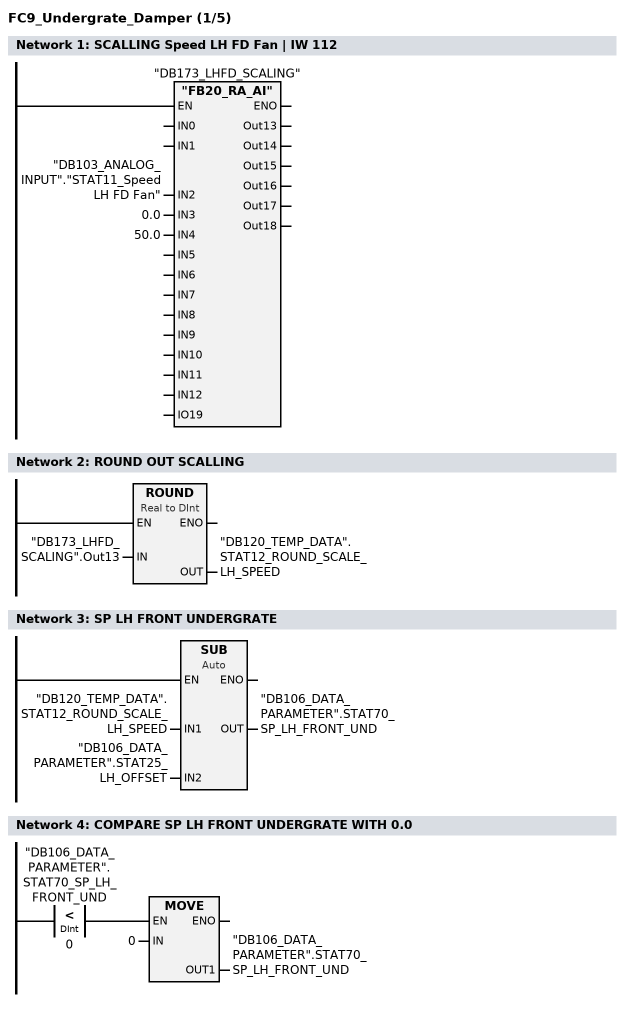
   RUNG wire#powerrail
      "DB173_LHFD_SCALING"(IN0 :=, IN1 :=, IN2 := "DB103_ANALOG_INPUT"."STAT11_Speed LH FD Fan", IN3 := 0.0, IN4 := 50.0, IN5 :=, IN6 :=, IN7 :=, IN8 :=, IN9 :=, IN10 :=, IN11 :=, IN12 :=, Out13 =>, IO19 :=, Out14 =>, Out15 =>, Out16 =>, Out17 =>, Out18 =>)
   END_RUNG
   // the same network as SCL:
   "DB173_LHFD_SCALING"(IN2 := "DB103_ANALOG_INPUT"."STAT11_Speed LH FD Fan", IN3 := 0.0, IN4 := 50.0);   // "FB20_RA_AI"
END_REGION

REGION Network 2: ROUND OUT SCALLING
   RUNG wire#powerrail
      { S7_Templates := "[SrcType := Real, DestType := DInt]" } Round(in := "DB173_LHFD_SCALING".Out13, out => "DB120_TEMP_DATA".STAT12_ROUND_SCALE_LH_SPEED)
   END_RUNG
   // the same network as SCL:
   "DB120_TEMP_DATA".STAT12_ROUND_SCALE_LH_SPEED := ROUND("DB173_LHFD_SCALING".Out13);
END_REGION

REGION Network 3: SP LH FRONT UNDERGRATE
   RUNG wire#powerrail
      Sub(in1 := "DB120_TEMP_DATA".STAT12_ROUND_SCALE_LH_SPEED, in2 := "DB106_DATA_PARAMETER".STAT25_LH_OFFSET, out => "DB106_DATA_PARAMETER".STAT70_SP_LH_FRONT_UND)
   END_RUNG
   // the same network as SCL:
   "DB106_DATA_PARAMETER".STAT70_SP_LH_FRONT_UND := "DB120_TEMP_DATA".STAT12_ROUND_SCALE_LH_SPEED - "DB106_DATA_PARAMETER".STAT25_LH_OFFSET;
END_REGION

REGION Network 4: COMPARE SP LH FRONT UNDERGRATE WITH 0.0
   RUNG wire#powerrail
      { S7_Templates := "SrcType := DInt" } LT_Contact(in1 := "DB106_DATA_PARAMETER".STAT70_SP_LH_FRONT_UND, in2 := 0)
      Move(in := 0, out1 => "DB106_DATA_PARAMETER".STAT70_SP_LH_FRONT_UND)
   END_RUNG
   // the same network as SCL:
   IF "DB106_DATA_PARAMETER".STAT70_SP_LH_FRONT_UND < 0 THEN
       "DB106_DATA_PARAMETER".STAT70_SP_LH_FRONT_UND := 0;
   END_IF;
END_REGION

REGION Network 5: LH FRONT UNDERGRATE POSITION | IW 208
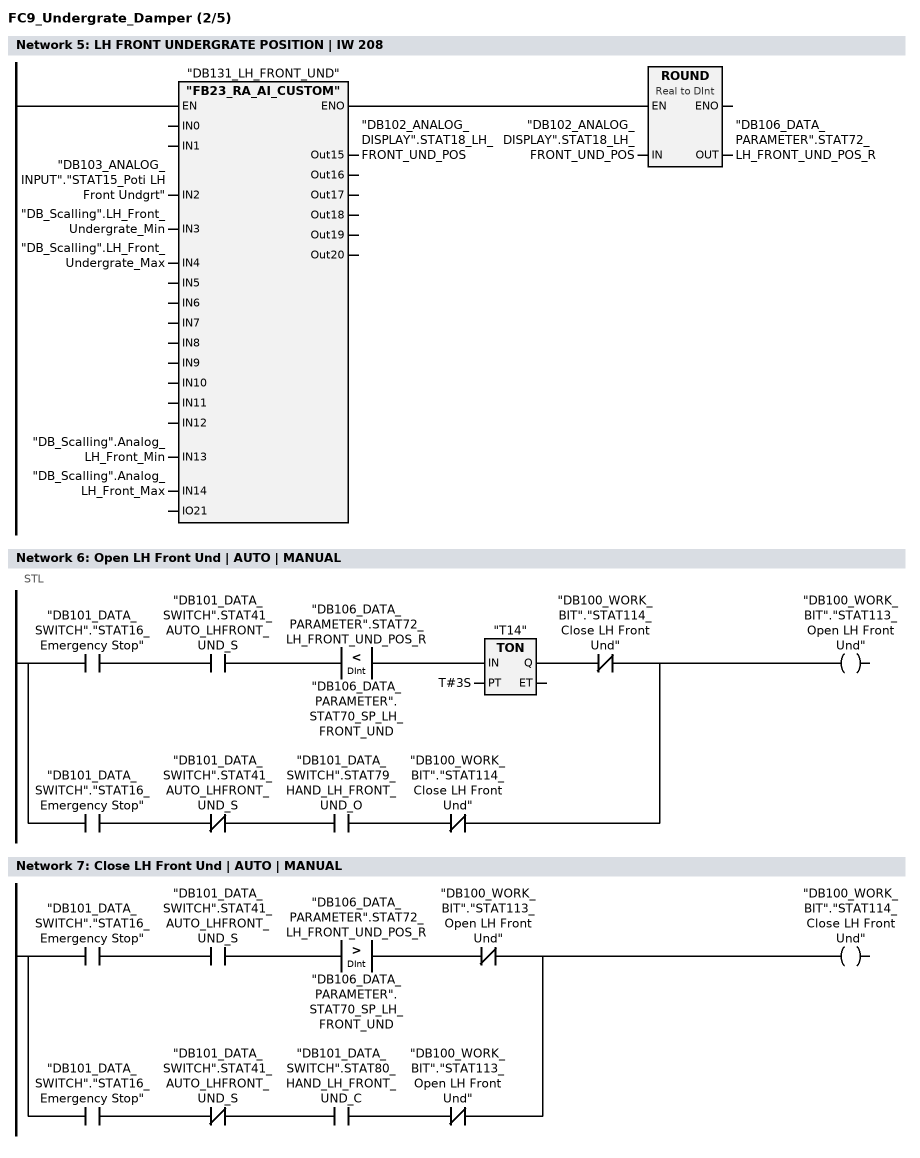
   RUNG wire#powerrail
      "DB131_LH_FRONT_UND"(IN0 :=, IN1 :=, IN2 := "DB103_ANALOG_INPUT"."STAT15_Poti LH Front Undgrt", IN3 := "DB_Scalling".LH_Front_Undergrate_Min, IN4 := "DB_Scalling".LH_Front_Undergrate_Max, IN5 :=, IN6 :=, IN7 :=, IN8 :=, IN9 :=, IN10 :=, IN11 :=, IN12 :=, IN13 := "DB_Scalling".Analog_LH_Front_Min, IN14 := "DB_Scalling".Analog_LH_Front_Max, IO21 :=, Out15 => "DB102_ANALOG_DISPLAY".STAT18_LH_FRONT_UND_POS, Out16 =>, Out17 =>, Out18 =>, Out19 =>, Out20 =>)
      { S7_Templates := "[SrcType := Real, DestType := DInt]" } Round(in := "DB102_ANALOG_DISPLAY".STAT18_LH_FRONT_UND_POS, out => "DB106_DATA_PARAMETER".STAT72_LH_FRONT_UND_POS_R)
   END_RUNG
   // the same network as SCL:
   "DB131_LH_FRONT_UND"(IN2 := "DB103_ANALOG_INPUT"."STAT15_Poti LH Front Undgrt",   // "FB23_RA_AI_CUSTOM"
                        IN3 := "DB_Scalling".LH_Front_Undergrate_Min,
                        IN4 := "DB_Scalling".LH_Front_Undergrate_Max,
                        IN13 := "DB_Scalling".Analog_LH_Front_Min,
                        IN14 := "DB_Scalling".Analog_LH_Front_Max,
                        Out15 => "DB102_ANALOG_DISPLAY".STAT18_LH_FRONT_UND_POS,
                        ENO => #_w1);
   IF #_w1 THEN
       "DB106_DATA_PARAMETER".STAT72_LH_FRONT_UND_POS_R := ROUND("DB102_ANALOG_DISPLAY".STAT18_LH_FRONT_UND_POS);
   END_IF;
END_REGION

REGION Network 6: Open LH Front Und | AUTO | MANUAL
   // STL
   "T14".TON(IN := "DB101_DATA_SWITCH"."STAT16_Emergency Stop" AND "DB101_DATA_SWITCH".STAT41_AUTO_LHFRONT_UND_S AND ("DB106_DATA_PARAMETER".STAT72_LH_FRONT_UND_POS_R < "DB106_DATA_PARAMETER".STAT70_SP_LH_FRONT_UND),
             PT := T#3S);
   "DB100_WORK_BIT"."STAT113_Open LH Front Und" := ("T14".Q AND NOT "DB100_WORK_BIT"."STAT114_Close LH Front Und") OR ("DB101_DATA_SWITCH"."STAT16_Emergency Stop" AND NOT "DB101_DATA_SWITCH".STAT41_AUTO_LHFRONT_UND_S AND "DB101_DATA_SWITCH".STAT79_HAND_LH_FRONT_UND_O AND NOT "DB100_WORK_BIT"."STAT114_Close LH Front Und");
END_REGION

REGION Network 7: Close LH Front Und | AUTO | MANUAL
   RUNG wire#powerrail
      Contact( "DB101_DATA_SWITCH"."STAT16_Emergency Stop" )
      Contact( "DB101_DATA_SWITCH".STAT41_AUTO_LHFRONT_UND_S )
      { S7_Templates := "SrcType := DInt" } GT_Contact(in1 := "DB106_DATA_PARAMETER".STAT72_LH_FRONT_UND_POS_R, in2 := "DB106_DATA_PARAMETER".STAT70_SP_LH_FRONT_UND)
      I_Contact( "DB100_WORK_BIT"."STAT113_Open LH Front Und" )
      wire#w1
      Coil( "DB100_WORK_BIT"."STAT114_Close LH Front Und" )
   END_RUNG
   RUNG wire#powerrail
      Contact( "DB101_DATA_SWITCH"."STAT16_Emergency Stop" )
      I_Contact( "DB101_DATA_SWITCH".STAT41_AUTO_LHFRONT_UND_S )
      Contact( "DB101_DATA_SWITCH".STAT80_HAND_LH_FRONT_UND_C )
      I_Contact( "DB100_WORK_BIT"."STAT113_Open LH Front Und" )
   END_RUNG wire#w1
   // the same network as SCL:
   "DB100_WORK_BIT"."STAT114_Close LH Front Und" := ("DB101_DATA_SWITCH"."STAT16_Emergency Stop" AND "DB101_DATA_SWITCH".STAT41_AUTO_LHFRONT_UND_S AND ("DB106_DATA_PARAMETER".STAT72_LH_FRONT_UND_POS_R > "DB106_DATA_PARAMETER".STAT70_SP_LH_FRONT_UND) AND NOT "DB100_WORK_BIT"."STAT113_Open LH Front Und") OR ("DB101_DATA_SWITCH"."STAT16_Emergency Stop" AND NOT "DB101_DATA_SWITCH".STAT41_AUTO_LHFRONT_UND_S AND "DB101_DATA_SWITCH".STAT80_HAND_LH_FRONT_UND_C AND NOT "DB100_WORK_BIT"."STAT113_Open LH Front Und");
END_REGION

REGION Network 8: SCALLING Speed RH FD Fan | IW 114
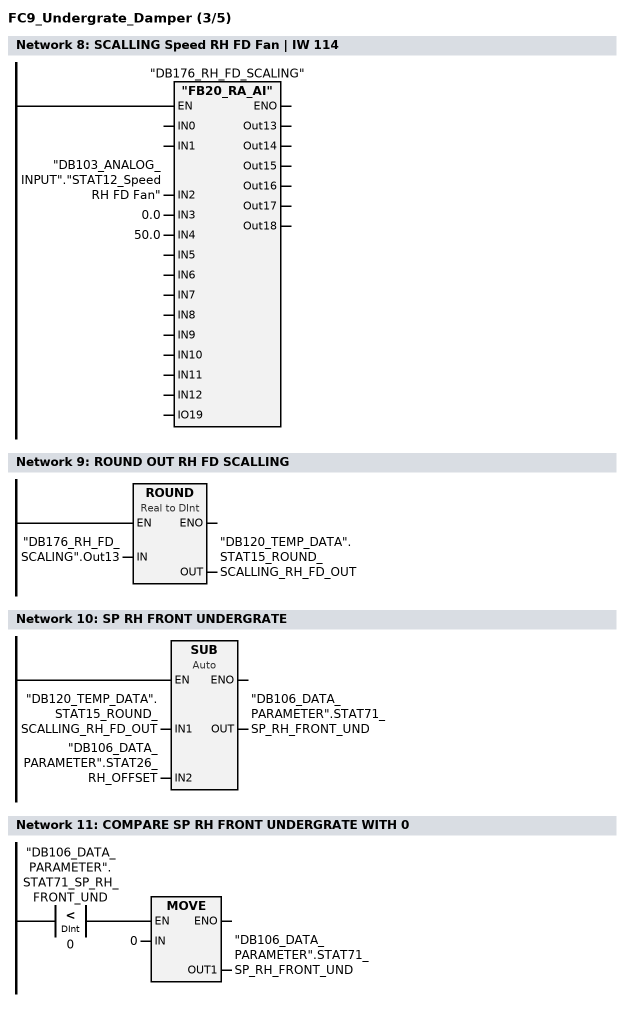
   RUNG wire#powerrail
      "DB176_RH_FD_SCALING"(IN0 :=, IN1 :=, IN2 := "DB103_ANALOG_INPUT"."STAT12_Speed RH FD Fan", IN3 := 0.0, IN4 := 50.0, IN5 :=, IN6 :=, IN7 :=, IN8 :=, IN9 :=, IN10 :=, IN11 :=, IN12 :=, Out13 =>, IO19 :=, Out14 =>, Out15 =>, Out16 =>, Out17 =>, Out18 =>)
   END_RUNG
   // the same network as SCL:
   "DB176_RH_FD_SCALING"(IN2 := "DB103_ANALOG_INPUT"."STAT12_Speed RH FD Fan", IN3 := 0.0, IN4 := 50.0);   // "FB20_RA_AI"
END_REGION

REGION Network 9: ROUND OUT RH FD SCALLING
   RUNG wire#powerrail
      { S7_Templates := "[SrcType := Real, DestType := DInt]" } Round(in := "DB176_RH_FD_SCALING".Out13, out => "DB120_TEMP_DATA".STAT15_ROUND_SCALLING_RH_FD_OUT)
   END_RUNG
   // the same network as SCL:
   "DB120_TEMP_DATA".STAT15_ROUND_SCALLING_RH_FD_OUT := ROUND("DB176_RH_FD_SCALING".Out13);
END_REGION

REGION Network 10: SP RH FRONT UNDERGRATE
   RUNG wire#powerrail
      Sub(in1 := "DB120_TEMP_DATA".STAT15_ROUND_SCALLING_RH_FD_OUT, in2 := "DB106_DATA_PARAMETER".STAT26_RH_OFFSET, out => "DB106_DATA_PARAMETER".STAT71_SP_RH_FRONT_UND)
   END_RUNG
   // the same network as SCL:
   "DB106_DATA_PARAMETER".STAT71_SP_RH_FRONT_UND := "DB120_TEMP_DATA".STAT15_ROUND_SCALLING_RH_FD_OUT - "DB106_DATA_PARAMETER".STAT26_RH_OFFSET;
END_REGION

REGION Network 11: COMPARE SP RH FRONT UNDERGRATE WITH 0
   RUNG wire#powerrail
      { S7_Templates := "SrcType := DInt" } LT_Contact(in1 := "DB106_DATA_PARAMETER".STAT71_SP_RH_FRONT_UND, in2 := 0)
      Move(in := 0, out1 => "DB106_DATA_PARAMETER".STAT71_SP_RH_FRONT_UND)
   END_RUNG
   // the same network as SCL:
   IF "DB106_DATA_PARAMETER".STAT71_SP_RH_FRONT_UND < 0 THEN
       "DB106_DATA_PARAMETER".STAT71_SP_RH_FRONT_UND := 0;
   END_IF;
END_REGION

REGION Network 12: Poti RH Front Undgrt(FEED BACK POSITION) RH FRONT UNDERGRATE
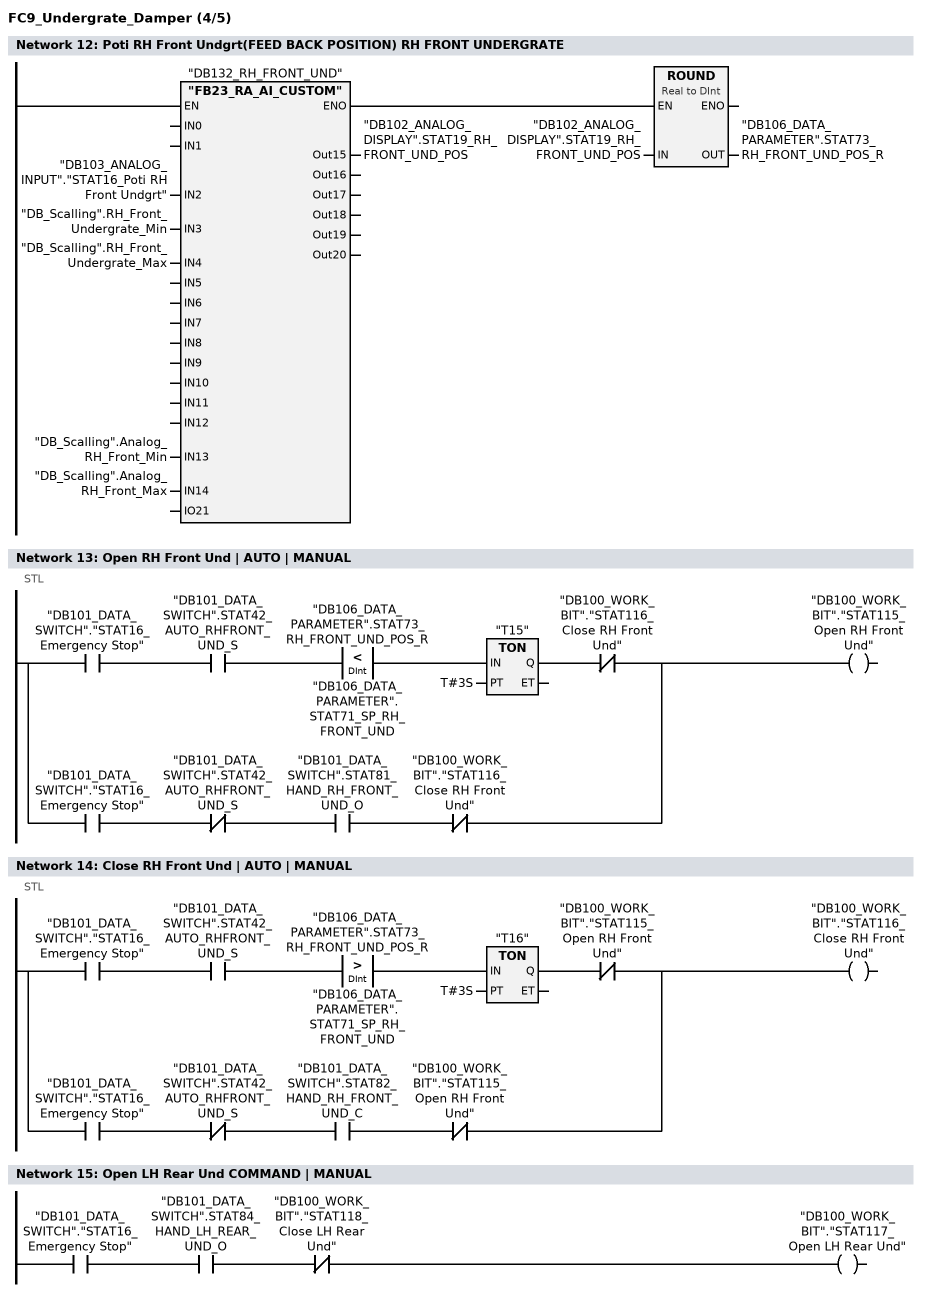
   RUNG wire#powerrail
      "DB132_RH_FRONT_UND"(IN0 :=, IN1 :=, IN2 := "DB103_ANALOG_INPUT"."STAT16_Poti RH Front Undgrt", IN3 := "DB_Scalling".RH_Front_Undergrate_Min, IN4 := "DB_Scalling".RH_Front_Undergrate_Max, IN5 :=, IN6 :=, IN7 :=, IN8 :=, IN9 :=, IN10 :=, IN11 :=, IN12 :=, IN13 := "DB_Scalling".Analog_RH_Front_Min, IN14 := "DB_Scalling".Analog_RH_Front_Max, IO21 :=, Out15 => "DB102_ANALOG_DISPLAY".STAT19_RH_FRONT_UND_POS, Out16 =>, Out17 =>, Out18 =>, Out19 =>, Out20 =>)
      { S7_Templates := "[SrcType := Real, DestType := DInt]" } Round(in := "DB102_ANALOG_DISPLAY".STAT19_RH_FRONT_UND_POS, out => "DB106_DATA_PARAMETER".STAT73_RH_FRONT_UND_POS_R)
   END_RUNG
   // the same network as SCL:
   "DB132_RH_FRONT_UND"(IN2 := "DB103_ANALOG_INPUT"."STAT16_Poti RH Front Undgrt",   // "FB23_RA_AI_CUSTOM"
                        IN3 := "DB_Scalling".RH_Front_Undergrate_Min,
                        IN4 := "DB_Scalling".RH_Front_Undergrate_Max,
                        IN13 := "DB_Scalling".Analog_RH_Front_Min,
                        IN14 := "DB_Scalling".Analog_RH_Front_Max,
                        Out15 => "DB102_ANALOG_DISPLAY".STAT19_RH_FRONT_UND_POS,
                        ENO => #_w1);
   IF #_w1 THEN
       "DB106_DATA_PARAMETER".STAT73_RH_FRONT_UND_POS_R := ROUND("DB102_ANALOG_DISPLAY".STAT19_RH_FRONT_UND_POS);
   END_IF;
END_REGION

REGION Network 13: Open RH Front Und | AUTO | MANUAL
   // STL
   "T15".TON(IN := "DB101_DATA_SWITCH"."STAT16_Emergency Stop" AND "DB101_DATA_SWITCH".STAT42_AUTO_RHFRONT_UND_S AND ("DB106_DATA_PARAMETER".STAT73_RH_FRONT_UND_POS_R < "DB106_DATA_PARAMETER".STAT71_SP_RH_FRONT_UND),
             PT := T#3S);
   "DB100_WORK_BIT"."STAT115_Open RH Front Und" := ("T15".Q AND NOT "DB100_WORK_BIT"."STAT116_Close RH Front Und") OR ("DB101_DATA_SWITCH"."STAT16_Emergency Stop" AND NOT "DB101_DATA_SWITCH".STAT42_AUTO_RHFRONT_UND_S AND "DB101_DATA_SWITCH".STAT81_HAND_RH_FRONT_UND_O AND NOT "DB100_WORK_BIT"."STAT116_Close RH Front Und");
END_REGION

REGION Network 14: Close RH Front Und | AUTO | MANUAL
   // STL
   "T16".TON(IN := "DB101_DATA_SWITCH"."STAT16_Emergency Stop" AND "DB101_DATA_SWITCH".STAT42_AUTO_RHFRONT_UND_S AND ("DB106_DATA_PARAMETER".STAT73_RH_FRONT_UND_POS_R > "DB106_DATA_PARAMETER".STAT71_SP_RH_FRONT_UND),
             PT := T#3S);
   "DB100_WORK_BIT"."STAT116_Close RH Front Und" := ("T16".Q AND NOT "DB100_WORK_BIT"."STAT115_Open RH Front Und") OR ("DB101_DATA_SWITCH"."STAT16_Emergency Stop" AND NOT "DB101_DATA_SWITCH".STAT42_AUTO_RHFRONT_UND_S AND "DB101_DATA_SWITCH".STAT82_HAND_RH_FRONT_UND_C AND NOT "DB100_WORK_BIT"."STAT115_Open RH Front Und");
END_REGION

REGION Network 15: Open LH Rear Und COMMAND | MANUAL
   RUNG wire#powerrail
      Contact( "DB101_DATA_SWITCH"."STAT16_Emergency Stop" )
      Contact( "DB101_DATA_SWITCH".STAT84_HAND_LH_REAR_UND_O )
      I_Contact( "DB100_WORK_BIT"."STAT118_Close LH Rear Und" )
      Coil( "DB100_WORK_BIT"."STAT117_Open LH Rear Und" )
   END_RUNG
   // the same network as SCL:
   "DB100_WORK_BIT"."STAT117_Open LH Rear Und" := "DB101_DATA_SWITCH"."STAT16_Emergency Stop" AND "DB101_DATA_SWITCH".STAT84_HAND_LH_REAR_UND_O AND NOT "DB100_WORK_BIT"."STAT118_Close LH Rear Und";
END_REGION

REGION Network 16: Close LH Rear Und COMMAND | MANUAL
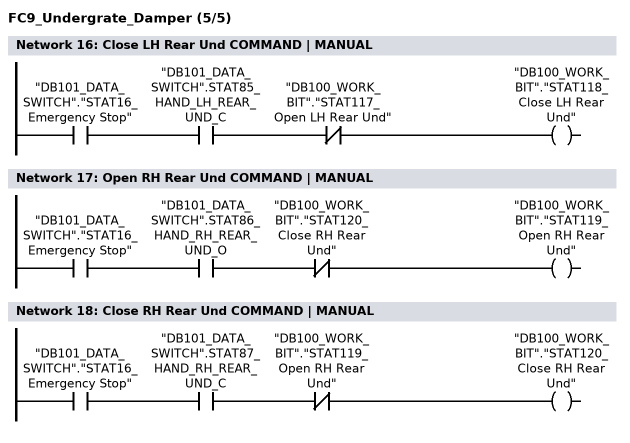
   RUNG wire#powerrail
      Contact( "DB101_DATA_SWITCH"."STAT16_Emergency Stop" )
      Contact( "DB101_DATA_SWITCH".STAT85_HAND_LH_REAR_UND_C )
      I_Contact( "DB100_WORK_BIT"."STAT117_Open LH Rear Und" )
      Coil( "DB100_WORK_BIT"."STAT118_Close LH Rear Und" )
   END_RUNG
   // the same network as SCL:
   "DB100_WORK_BIT"."STAT118_Close LH Rear Und" := "DB101_DATA_SWITCH"."STAT16_Emergency Stop" AND "DB101_DATA_SWITCH".STAT85_HAND_LH_REAR_UND_C AND NOT "DB100_WORK_BIT"."STAT117_Open LH Rear Und";
END_REGION

REGION Network 17: Open RH Rear Und COMMAND | MANUAL
   RUNG wire#powerrail
      Contact( "DB101_DATA_SWITCH"."STAT16_Emergency Stop" )
      Contact( "DB101_DATA_SWITCH".STAT86_HAND_RH_REAR_UND_O )
      I_Contact( "DB100_WORK_BIT"."STAT120_Close RH Rear Und" )
      Coil( "DB100_WORK_BIT"."STAT119_Open RH Rear Und" )
   END_RUNG
   // the same network as SCL:
   "DB100_WORK_BIT"."STAT119_Open RH Rear Und" := "DB101_DATA_SWITCH"."STAT16_Emergency Stop" AND "DB101_DATA_SWITCH".STAT86_HAND_RH_REAR_UND_O AND NOT "DB100_WORK_BIT"."STAT120_Close RH Rear Und";
END_REGION

REGION Network 18: Close RH Rear Und COMMAND | MANUAL
   RUNG wire#powerrail
      Contact( "DB101_DATA_SWITCH"."STAT16_Emergency Stop" )
      Contact( "DB101_DATA_SWITCH".STAT87_HAND_RH_REAR_UND_C )
      I_Contact( "DB100_WORK_BIT"."STAT119_Open RH Rear Und" )
      Coil( "DB100_WORK_BIT"."STAT120_Close RH Rear Und" )
   END_RUNG
   // the same network as SCL:
   "DB100_WORK_BIT"."STAT120_Close RH Rear Und" := "DB101_DATA_SWITCH"."STAT16_Emergency Stop" AND "DB101_DATA_SWITCH".STAT87_HAND_RH_REAR_UND_C AND NOT "DB100_WORK_BIT"."STAT119_Open RH Rear Und";
END_REGION
END_FUNCTION

FUNCTION "FC10_COAL_COUNTER" : Void   // FC10, LAD
TITLE = COAL COUNTER
{ S7_Optimized_Access := 'TRUE' }
VERSION : 0.1
BEGIN

REGION Network 1: LH TOTAL COAL
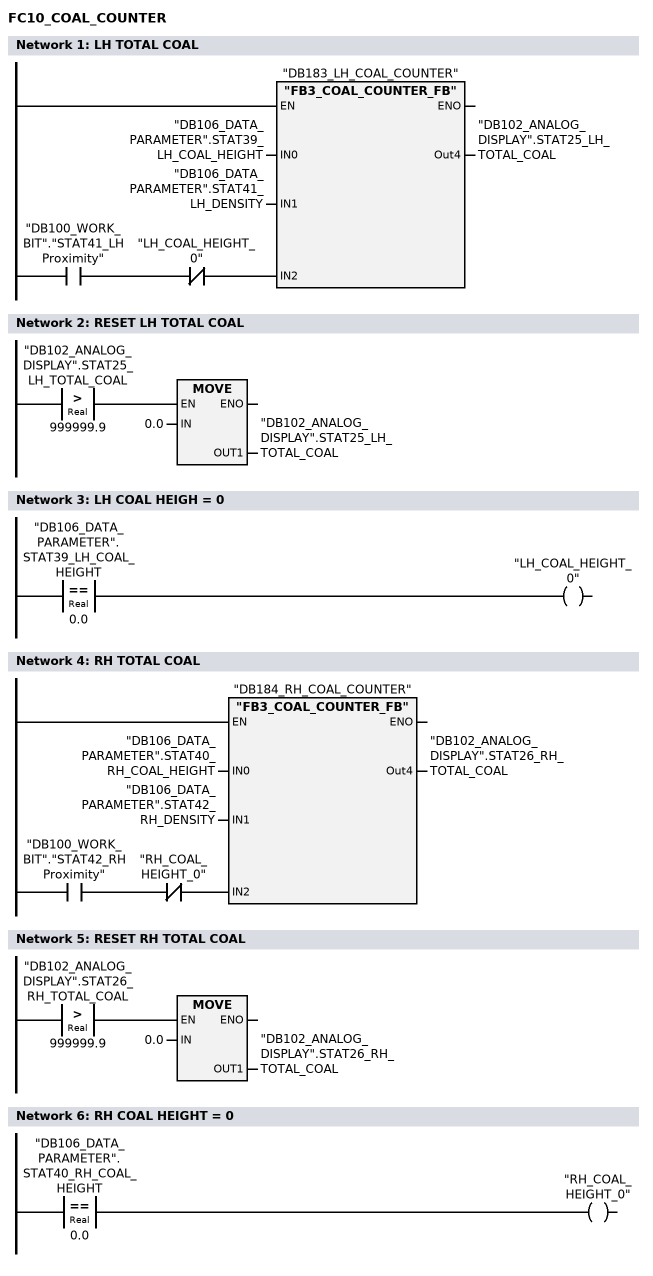
   RUNG wire#powerrail
      "DB183_LH_COAL_COUNTER"(IN2 := wire#w1, IN0 := "DB106_DATA_PARAMETER".STAT39_LH_COAL_HEIGHT, IN1 := "DB106_DATA_PARAMETER".STAT41_LH_DENSITY, Out4 => "DB102_ANALOG_DISPLAY".STAT25_LH_TOTAL_COAL)
   END_RUNG
   RUNG wire#powerrail
      Contact( "DB100_WORK_BIT"."STAT41_LH Proximity" )
      I_Contact( "LH_COAL_HEIGHT_0" )
   END_RUNG wire#w1
   // the same network as SCL:
   "DB183_LH_COAL_COUNTER"(IN0 := "DB106_DATA_PARAMETER".STAT39_LH_COAL_HEIGHT,   // "FB3_COAL_COUNTER_FB"
                           IN1 := "DB106_DATA_PARAMETER".STAT41_LH_DENSITY,
                           IN2 := "DB100_WORK_BIT"."STAT41_LH Proximity" AND NOT "LH_COAL_HEIGHT_0",
                           Out4 => "DB102_ANALOG_DISPLAY".STAT25_LH_TOTAL_COAL);
END_REGION

REGION Network 2: RESET LH TOTAL COAL
   RUNG wire#powerrail
      { S7_Templates := "SrcType := Real" } GT_Contact(in1 := "DB102_ANALOG_DISPLAY".STAT25_LH_TOTAL_COAL, in2 := 999999.9)
      Move(in := 0.0, out1 => "DB102_ANALOG_DISPLAY".STAT25_LH_TOTAL_COAL)
   END_RUNG
   // the same network as SCL:
   IF "DB102_ANALOG_DISPLAY".STAT25_LH_TOTAL_COAL > 999999.9 THEN
       "DB102_ANALOG_DISPLAY".STAT25_LH_TOTAL_COAL := 0.0;
   END_IF;
END_REGION

REGION Network 3: LH COAL HEIGH = 0
   RUNG wire#powerrail
      { S7_Templates := "SrcType := Real" } EQ_Contact(in1 := "DB106_DATA_PARAMETER".STAT39_LH_COAL_HEIGHT, in2 := 0.0)
      Coil( "LH_COAL_HEIGHT_0" )
   END_RUNG
   // the same network as SCL:
   "LH_COAL_HEIGHT_0" := "DB106_DATA_PARAMETER".STAT39_LH_COAL_HEIGHT = 0.0;
END_REGION

REGION Network 4: RH TOTAL COAL
   RUNG wire#powerrail
      "DB184_RH_COAL_COUNTER"(IN2 := wire#w1, IN0 := "DB106_DATA_PARAMETER".STAT40_RH_COAL_HEIGHT, IN1 := "DB106_DATA_PARAMETER".STAT42_RH_DENSITY, Out4 => "DB102_ANALOG_DISPLAY".STAT26_RH_TOTAL_COAL)
   END_RUNG
   RUNG wire#powerrail
      Contact( "DB100_WORK_BIT"."STAT42_RH Proximity" )
      I_Contact( "RH_COAL_HEIGHT_0" )
   END_RUNG wire#w1
   // the same network as SCL:
   "DB184_RH_COAL_COUNTER"(IN0 := "DB106_DATA_PARAMETER".STAT40_RH_COAL_HEIGHT,   // "FB3_COAL_COUNTER_FB"
                           IN1 := "DB106_DATA_PARAMETER".STAT42_RH_DENSITY,
                           IN2 := "DB100_WORK_BIT"."STAT42_RH Proximity" AND NOT "RH_COAL_HEIGHT_0",
                           Out4 => "DB102_ANALOG_DISPLAY".STAT26_RH_TOTAL_COAL);
END_REGION

REGION Network 5: RESET RH TOTAL COAL
   RUNG wire#powerrail
      { S7_Templates := "SrcType := Real" } GT_Contact(in1 := "DB102_ANALOG_DISPLAY".STAT26_RH_TOTAL_COAL, in2 := 999999.9)
      Move(in := 0.0, out1 => "DB102_ANALOG_DISPLAY".STAT26_RH_TOTAL_COAL)
   END_RUNG
   // the same network as SCL:
   IF "DB102_ANALOG_DISPLAY".STAT26_RH_TOTAL_COAL > 999999.9 THEN
       "DB102_ANALOG_DISPLAY".STAT26_RH_TOTAL_COAL := 0.0;
   END_IF;
END_REGION

REGION Network 6: RH COAL HEIGHT = 0
   RUNG wire#powerrail
      { S7_Templates := "SrcType := Real" } EQ_Contact(in1 := "DB106_DATA_PARAMETER".STAT40_RH_COAL_HEIGHT, in2 := 0.0)
      Coil( "RH_COAL_HEIGHT_0" )
   END_RUNG
   // the same network as SCL:
   "RH_COAL_HEIGHT_0" := "DB106_DATA_PARAMETER".STAT40_RH_COAL_HEIGHT = 0.0;
END_REGION
END_FUNCTION

FUNCTION "FC11_Alarm" : Void   // FC11, LAD
TITLE = ALARM
{ S7_Optimized_Access := 'TRUE' }
VERSION : 0.1
BEGIN

REGION Network 1: Alarm Low Water PreWarning
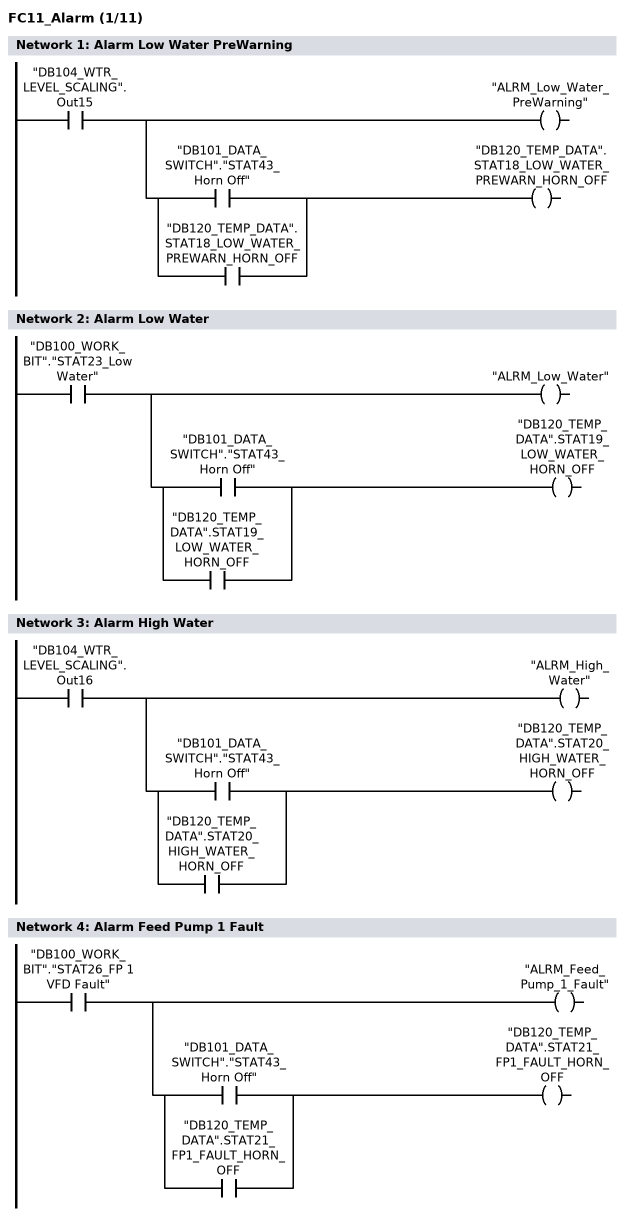
   RUNG wire#powerrail
      Contact( "DB104_WTR_LEVEL_SCALING".Out15 )
      wire#w1
      Coil( "ALRM_Low_Water_PreWarning" )
   END_RUNG
   RUNG wire#w1
      Contact( "DB101_DATA_SWITCH"."STAT43_Horn Off" )
      wire#w2
      Coil( "DB120_TEMP_DATA".STAT18_LOW_WATER_PREWARN_HORN_OFF )
   END_RUNG
   RUNG wire#w1
      Contact( "DB120_TEMP_DATA".STAT18_LOW_WATER_PREWARN_HORN_OFF )
   END_RUNG wire#w2
   // the same network as SCL:
   "ALRM_Low_Water_PreWarning" := "DB104_WTR_LEVEL_SCALING".Out15;
   "DB120_TEMP_DATA".STAT18_LOW_WATER_PREWARN_HORN_OFF := "DB104_WTR_LEVEL_SCALING".Out15 AND ("DB101_DATA_SWITCH"."STAT43_Horn Off" OR "DB120_TEMP_DATA".STAT18_LOW_WATER_PREWARN_HORN_OFF);
END_REGION

REGION Network 2: Alarm Low Water
   RUNG wire#powerrail
      Contact( "DB100_WORK_BIT"."STAT23_Low Water" )
      wire#w1
      Coil( "ALRM_Low_Water" )
   END_RUNG
   RUNG wire#w1
      Contact( "DB101_DATA_SWITCH"."STAT43_Horn Off" )
      wire#w2
      Coil( "DB120_TEMP_DATA".STAT19_LOW_WATER_HORN_OFF )
   END_RUNG
   RUNG wire#w1
      Contact( "DB120_TEMP_DATA".STAT19_LOW_WATER_HORN_OFF )
   END_RUNG wire#w2
   // the same network as SCL:
   "ALRM_Low_Water" := "DB100_WORK_BIT"."STAT23_Low Water";
   "DB120_TEMP_DATA".STAT19_LOW_WATER_HORN_OFF := "DB100_WORK_BIT"."STAT23_Low Water" AND ("DB101_DATA_SWITCH"."STAT43_Horn Off" OR "DB120_TEMP_DATA".STAT19_LOW_WATER_HORN_OFF);
END_REGION

REGION Network 3: Alarm High Water
   RUNG wire#powerrail
      Contact( "DB104_WTR_LEVEL_SCALING".Out16 )
      wire#w1
      Coil( "ALRM_High_Water" )
   END_RUNG
   RUNG wire#w1
      Contact( "DB101_DATA_SWITCH"."STAT43_Horn Off" )
      wire#w2
      Coil( "DB120_TEMP_DATA".STAT20_HIGH_WATER_HORN_OFF )
   END_RUNG
   RUNG wire#w1
      Contact( "DB120_TEMP_DATA".STAT20_HIGH_WATER_HORN_OFF )
   END_RUNG wire#w2
   // the same network as SCL:
   "ALRM_High_Water" := "DB104_WTR_LEVEL_SCALING".Out16;
   "DB120_TEMP_DATA".STAT20_HIGH_WATER_HORN_OFF := "DB104_WTR_LEVEL_SCALING".Out16 AND ("DB101_DATA_SWITCH"."STAT43_Horn Off" OR "DB120_TEMP_DATA".STAT20_HIGH_WATER_HORN_OFF);
END_REGION

REGION Network 4: Alarm Feed Pump 1 Fault
   RUNG wire#powerrail
      Contact( "DB100_WORK_BIT"."STAT26_FP 1 VFD Fault" )
      wire#w1
      Coil( "ALRM_Feed_Pump_1_Fault" )
   END_RUNG
   RUNG wire#w1
      Contact( "DB101_DATA_SWITCH"."STAT43_Horn Off" )
      wire#w2
      Coil( "DB120_TEMP_DATA".STAT21_FP1_FAULT_HORN_OFF )
   END_RUNG
   RUNG wire#w1
      Contact( "DB120_TEMP_DATA".STAT21_FP1_FAULT_HORN_OFF )
   END_RUNG wire#w2
   // the same network as SCL:
   "ALRM_Feed_Pump_1_Fault" := "DB100_WORK_BIT"."STAT26_FP 1 VFD Fault";
   "DB120_TEMP_DATA".STAT21_FP1_FAULT_HORN_OFF := "DB100_WORK_BIT"."STAT26_FP 1 VFD Fault" AND ("DB101_DATA_SWITCH"."STAT43_Horn Off" OR "DB120_TEMP_DATA".STAT21_FP1_FAULT_HORN_OFF);
END_REGION

REGION Network 5: Alarm Feed Pump 2 Fault
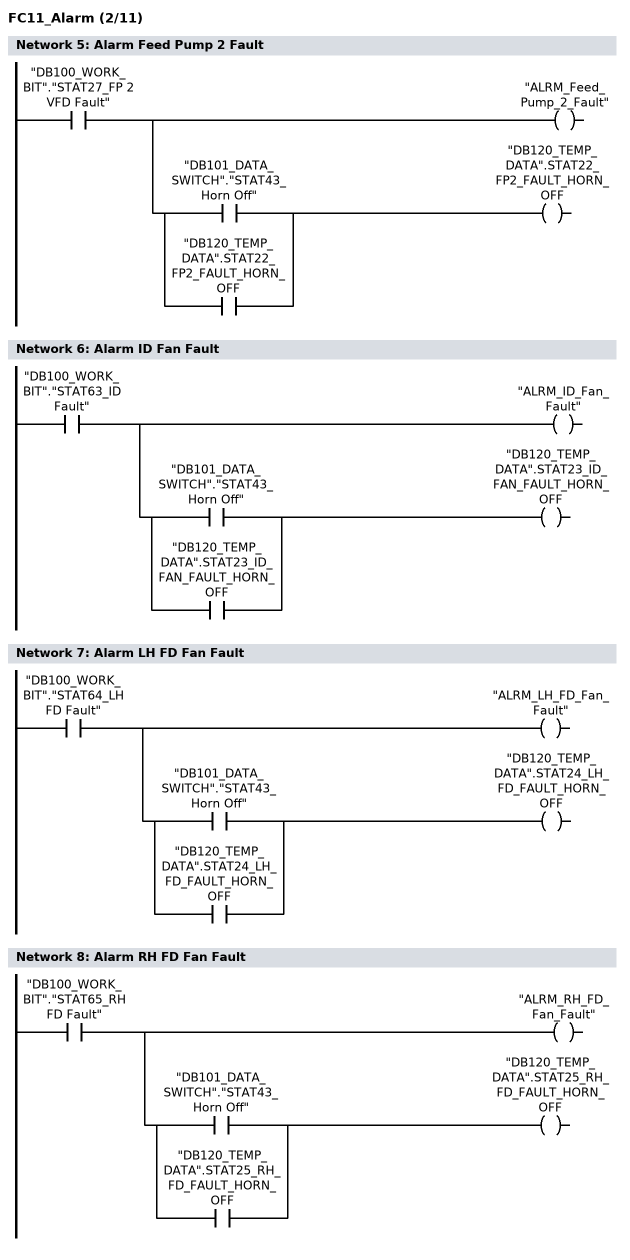
   RUNG wire#powerrail
      Contact( "DB100_WORK_BIT"."STAT27_FP 2 VFD Fault" )
      wire#w1
      Coil( "ALRM_Feed_Pump_2_Fault" )
   END_RUNG
   RUNG wire#w1
      Contact( "DB101_DATA_SWITCH"."STAT43_Horn Off" )
      wire#w2
      Coil( "DB120_TEMP_DATA".STAT22_FP2_FAULT_HORN_OFF )
   END_RUNG
   RUNG wire#w1
      Contact( "DB120_TEMP_DATA".STAT22_FP2_FAULT_HORN_OFF )
   END_RUNG wire#w2
   // the same network as SCL:
   "ALRM_Feed_Pump_2_Fault" := "DB100_WORK_BIT"."STAT27_FP 2 VFD Fault";
   "DB120_TEMP_DATA".STAT22_FP2_FAULT_HORN_OFF := "DB100_WORK_BIT"."STAT27_FP 2 VFD Fault" AND ("DB101_DATA_SWITCH"."STAT43_Horn Off" OR "DB120_TEMP_DATA".STAT22_FP2_FAULT_HORN_OFF);
END_REGION

REGION Network 6: Alarm ID Fan Fault
   RUNG wire#powerrail
      Contact( "DB100_WORK_BIT"."STAT63_ID Fault" )
      wire#w1
      Coil( "ALRM_ID_Fan_Fault" )
   END_RUNG
   RUNG wire#w1
      Contact( "DB101_DATA_SWITCH"."STAT43_Horn Off" )
      wire#w2
      Coil( "DB120_TEMP_DATA".STAT23_ID_FAN_FAULT_HORN_OFF )
   END_RUNG
   RUNG wire#w1
      Contact( "DB120_TEMP_DATA".STAT23_ID_FAN_FAULT_HORN_OFF )
   END_RUNG wire#w2
   // the same network as SCL:
   "ALRM_ID_Fan_Fault" := "DB100_WORK_BIT"."STAT63_ID Fault";
   "DB120_TEMP_DATA".STAT23_ID_FAN_FAULT_HORN_OFF := "DB100_WORK_BIT"."STAT63_ID Fault" AND ("DB101_DATA_SWITCH"."STAT43_Horn Off" OR "DB120_TEMP_DATA".STAT23_ID_FAN_FAULT_HORN_OFF);
END_REGION

REGION Network 7: Alarm LH FD Fan Fault
   RUNG wire#powerrail
      Contact( "DB100_WORK_BIT"."STAT64_LH FD Fault" )
      wire#w1
      Coil( "ALRM_LH_FD_Fan_Fault" )
   END_RUNG
   RUNG wire#w1
      Contact( "DB101_DATA_SWITCH"."STAT43_Horn Off" )
      wire#w2
      Coil( "DB120_TEMP_DATA".STAT24_LH_FD_FAULT_HORN_OFF )
   END_RUNG
   RUNG wire#w1
      Contact( "DB120_TEMP_DATA".STAT24_LH_FD_FAULT_HORN_OFF )
   END_RUNG wire#w2
   // the same network as SCL:
   "ALRM_LH_FD_Fan_Fault" := "DB100_WORK_BIT"."STAT64_LH FD Fault";
   "DB120_TEMP_DATA".STAT24_LH_FD_FAULT_HORN_OFF := "DB100_WORK_BIT"."STAT64_LH FD Fault" AND ("DB101_DATA_SWITCH"."STAT43_Horn Off" OR "DB120_TEMP_DATA".STAT24_LH_FD_FAULT_HORN_OFF);
END_REGION

REGION Network 8: Alarm RH FD Fan Fault
   RUNG wire#powerrail
      Contact( "DB100_WORK_BIT"."STAT65_RH FD Fault" )
      wire#w1
      Coil( "ALRM_RH_FD_Fan_Fault" )
   END_RUNG
   RUNG wire#w1
      Contact( "DB101_DATA_SWITCH"."STAT43_Horn Off" )
      wire#w2
      Coil( "DB120_TEMP_DATA".STAT25_RH_FD_FAULT_HORN_OFF )
   END_RUNG
   RUNG wire#w1
      Contact( "DB120_TEMP_DATA".STAT25_RH_FD_FAULT_HORN_OFF )
   END_RUNG wire#w2
   // the same network as SCL:
   "ALRM_RH_FD_Fan_Fault" := "DB100_WORK_BIT"."STAT65_RH FD Fault";
   "DB120_TEMP_DATA".STAT25_RH_FD_FAULT_HORN_OFF := "DB100_WORK_BIT"."STAT65_RH FD Fault" AND ("DB101_DATA_SWITCH"."STAT43_Horn Off" OR "DB120_TEMP_DATA".STAT25_RH_FD_FAULT_HORN_OFF);
END_REGION

REGION Network 9: Alarm LH Stoker Fault
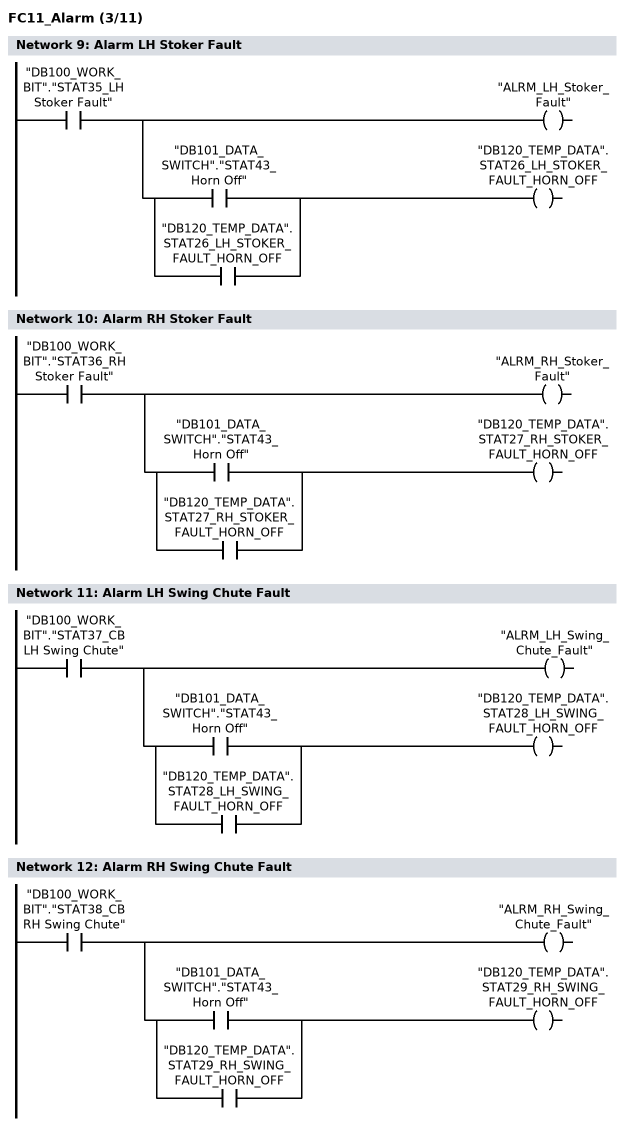
   RUNG wire#powerrail
      Contact( "DB100_WORK_BIT"."STAT35_LH Stoker Fault" )
      wire#w1
      Coil( "ALRM_LH_Stoker_Fault" )
   END_RUNG
   RUNG wire#w1
      Contact( "DB101_DATA_SWITCH"."STAT43_Horn Off" )
      wire#w2
      Coil( "DB120_TEMP_DATA".STAT26_LH_STOKER_FAULT_HORN_OFF )
   END_RUNG
   RUNG wire#w1
      Contact( "DB120_TEMP_DATA".STAT26_LH_STOKER_FAULT_HORN_OFF )
   END_RUNG wire#w2
   // the same network as SCL:
   "ALRM_LH_Stoker_Fault" := "DB100_WORK_BIT"."STAT35_LH Stoker Fault";
   "DB120_TEMP_DATA".STAT26_LH_STOKER_FAULT_HORN_OFF := "DB100_WORK_BIT"."STAT35_LH Stoker Fault" AND ("DB101_DATA_SWITCH"."STAT43_Horn Off" OR "DB120_TEMP_DATA".STAT26_LH_STOKER_FAULT_HORN_OFF);
END_REGION

REGION Network 10: Alarm RH Stoker Fault
   RUNG wire#powerrail
      Contact( "DB100_WORK_BIT"."STAT36_RH Stoker Fault" )
      wire#w1
      Coil( "ALRM_RH_Stoker_Fault" )
   END_RUNG
   RUNG wire#w1
      Contact( "DB101_DATA_SWITCH"."STAT43_Horn Off" )
      wire#w2
      Coil( "DB120_TEMP_DATA".STAT27_RH_STOKER_FAULT_HORN_OFF )
   END_RUNG
   RUNG wire#w1
      Contact( "DB120_TEMP_DATA".STAT27_RH_STOKER_FAULT_HORN_OFF )
   END_RUNG wire#w2
   // the same network as SCL:
   "ALRM_RH_Stoker_Fault" := "DB100_WORK_BIT"."STAT36_RH Stoker Fault";
   "DB120_TEMP_DATA".STAT27_RH_STOKER_FAULT_HORN_OFF := "DB100_WORK_BIT"."STAT36_RH Stoker Fault" AND ("DB101_DATA_SWITCH"."STAT43_Horn Off" OR "DB120_TEMP_DATA".STAT27_RH_STOKER_FAULT_HORN_OFF);
END_REGION

REGION Network 11: Alarm LH Swing Chute Fault
   RUNG wire#powerrail
      Contact( "DB100_WORK_BIT"."STAT37_CB LH Swing Chute" )
      wire#w1
      Coil( "ALRM_LH_Swing_Chute_Fault" )
   END_RUNG
   RUNG wire#w1
      Contact( "DB101_DATA_SWITCH"."STAT43_Horn Off" )
      wire#w2
      Coil( "DB120_TEMP_DATA".STAT28_LH_SWING_FAULT_HORN_OFF )
   END_RUNG
   RUNG wire#w1
      Contact( "DB120_TEMP_DATA".STAT28_LH_SWING_FAULT_HORN_OFF )
   END_RUNG wire#w2
   // the same network as SCL:
   "ALRM_LH_Swing_Chute_Fault" := "DB100_WORK_BIT"."STAT37_CB LH Swing Chute";
   "DB120_TEMP_DATA".STAT28_LH_SWING_FAULT_HORN_OFF := "DB100_WORK_BIT"."STAT37_CB LH Swing Chute" AND ("DB101_DATA_SWITCH"."STAT43_Horn Off" OR "DB120_TEMP_DATA".STAT28_LH_SWING_FAULT_HORN_OFF);
END_REGION

REGION Network 12: Alarm RH Swing Chute Fault
   RUNG wire#powerrail
      Contact( "DB100_WORK_BIT"."STAT38_CB RH Swing Chute" )
      wire#w1
      Coil( "ALRM_RH_Swing_Chute_Fault" )
   END_RUNG
   RUNG wire#w1
      Contact( "DB101_DATA_SWITCH"."STAT43_Horn Off" )
      wire#w2
      Coil( "DB120_TEMP_DATA".STAT29_RH_SWING_FAULT_HORN_OFF )
   END_RUNG
   RUNG wire#w1
      Contact( "DB120_TEMP_DATA".STAT29_RH_SWING_FAULT_HORN_OFF )
   END_RUNG wire#w2
   // the same network as SCL:
   "ALRM_RH_Swing_Chute_Fault" := "DB100_WORK_BIT"."STAT38_CB RH Swing Chute";
   "DB120_TEMP_DATA".STAT29_RH_SWING_FAULT_HORN_OFF := "DB100_WORK_BIT"."STAT38_CB RH Swing Chute" AND ("DB101_DATA_SWITCH"."STAT43_Horn Off" OR "DB120_TEMP_DATA".STAT29_RH_SWING_FAULT_HORN_OFF);
END_REGION

REGION Network 13: Alarm RAV1 Fault ASH VALVE 1
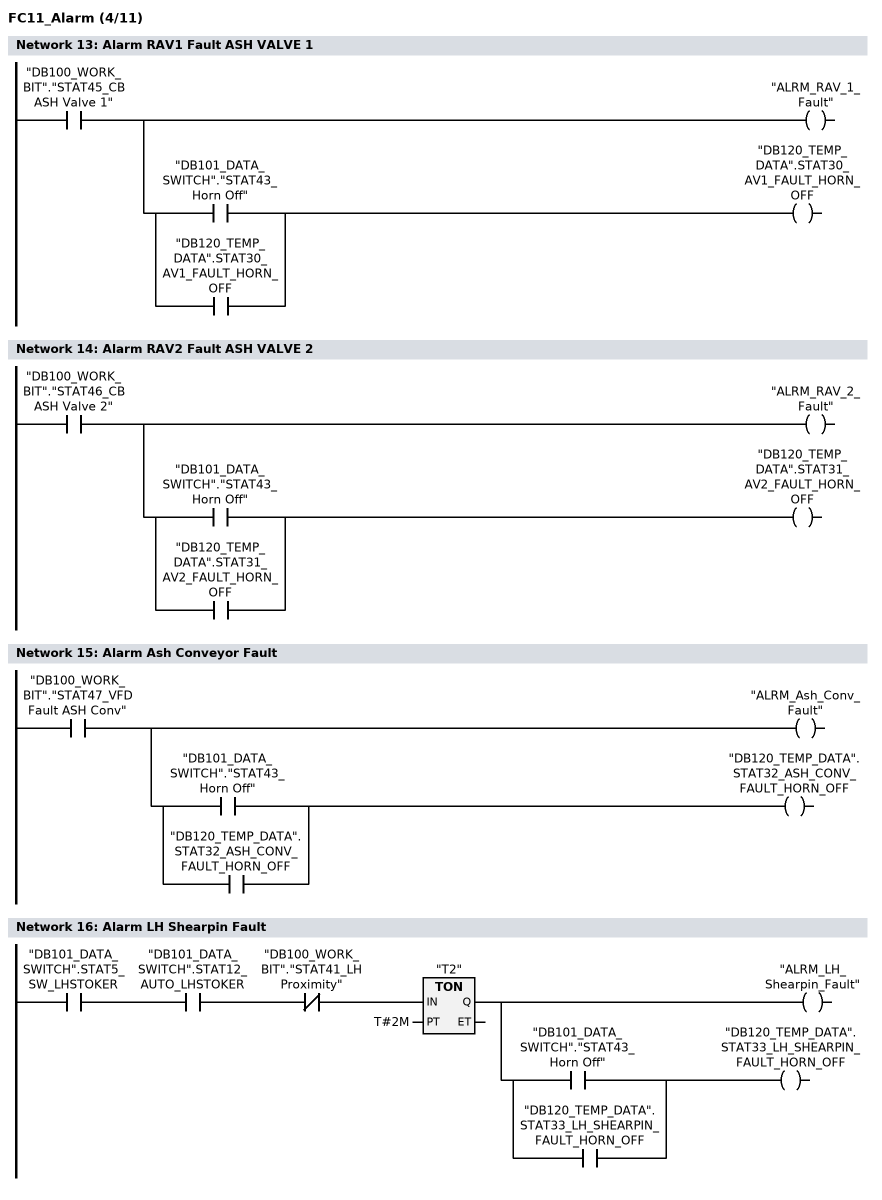
   RUNG wire#powerrail
      Contact( "DB100_WORK_BIT"."STAT45_CB ASH Valve 1" )
      wire#w1
      Coil( "ALRM_RAV_1_Fault" )
   END_RUNG
   RUNG wire#w1
      Contact( "DB101_DATA_SWITCH"."STAT43_Horn Off" )
      wire#w2
      Coil( "DB120_TEMP_DATA".STAT30_AV1_FAULT_HORN_OFF )
   END_RUNG
   RUNG wire#w1
      Contact( "DB120_TEMP_DATA".STAT30_AV1_FAULT_HORN_OFF )
   END_RUNG wire#w2
   // the same network as SCL:
   "ALRM_RAV_1_Fault" := "DB100_WORK_BIT"."STAT45_CB ASH Valve 1";
   "DB120_TEMP_DATA".STAT30_AV1_FAULT_HORN_OFF := "DB100_WORK_BIT"."STAT45_CB ASH Valve 1" AND ("DB101_DATA_SWITCH"."STAT43_Horn Off" OR "DB120_TEMP_DATA".STAT30_AV1_FAULT_HORN_OFF);
END_REGION

REGION Network 14: Alarm RAV2 Fault ASH VALVE 2
   RUNG wire#powerrail
      Contact( "DB100_WORK_BIT"."STAT46_CB ASH Valve 2" )
      wire#w1
      Coil( "ALRM_RAV_2_Fault" )
   END_RUNG
   RUNG wire#w1
      Contact( "DB101_DATA_SWITCH"."STAT43_Horn Off" )
      wire#w2
      Coil( "DB120_TEMP_DATA".STAT31_AV2_FAULT_HORN_OFF )
   END_RUNG
   RUNG wire#w1
      Contact( "DB120_TEMP_DATA".STAT31_AV2_FAULT_HORN_OFF )
   END_RUNG wire#w2
   // the same network as SCL:
   "ALRM_RAV_2_Fault" := "DB100_WORK_BIT"."STAT46_CB ASH Valve 2";
   "DB120_TEMP_DATA".STAT31_AV2_FAULT_HORN_OFF := "DB100_WORK_BIT"."STAT46_CB ASH Valve 2" AND ("DB101_DATA_SWITCH"."STAT43_Horn Off" OR "DB120_TEMP_DATA".STAT31_AV2_FAULT_HORN_OFF);
END_REGION

REGION Network 15: Alarm Ash Conveyor Fault
   RUNG wire#powerrail
      Contact( "DB100_WORK_BIT"."STAT47_VFD Fault ASH Conv" )
      wire#w1
      Coil( "ALRM_Ash_Conv_Fault" )
   END_RUNG
   RUNG wire#w1
      Contact( "DB101_DATA_SWITCH"."STAT43_Horn Off" )
      wire#w2
      Coil( "DB120_TEMP_DATA".STAT32_ASH_CONV_FAULT_HORN_OFF )
   END_RUNG
   RUNG wire#w1
      Contact( "DB120_TEMP_DATA".STAT32_ASH_CONV_FAULT_HORN_OFF )
   END_RUNG wire#w2
   // the same network as SCL:
   "ALRM_Ash_Conv_Fault" := "DB100_WORK_BIT"."STAT47_VFD Fault ASH Conv";
   "DB120_TEMP_DATA".STAT32_ASH_CONV_FAULT_HORN_OFF := "DB100_WORK_BIT"."STAT47_VFD Fault ASH Conv" AND ("DB101_DATA_SWITCH"."STAT43_Horn Off" OR "DB120_TEMP_DATA".STAT32_ASH_CONV_FAULT_HORN_OFF);
END_REGION

REGION Network 16: Alarm LH Shearpin Fault
   "T2".TON(IN := "DB101_DATA_SWITCH".STAT5_SW_LHSTOKER AND "DB101_DATA_SWITCH".STAT12_AUTO_LHSTOKER AND NOT "DB100_WORK_BIT"."STAT41_LH Proximity",
            PT := T#2M);
   "ALRM_LH_Shearpin_Fault" := "T2".Q;
   "DB120_TEMP_DATA".STAT33_LH_SHEARPIN_FAULT_HORN_OFF := "T2".Q AND ("DB101_DATA_SWITCH"."STAT43_Horn Off" OR "DB120_TEMP_DATA".STAT33_LH_SHEARPIN_FAULT_HORN_OFF);
END_REGION

REGION Network 17: Alarm RH Shearpin Fault
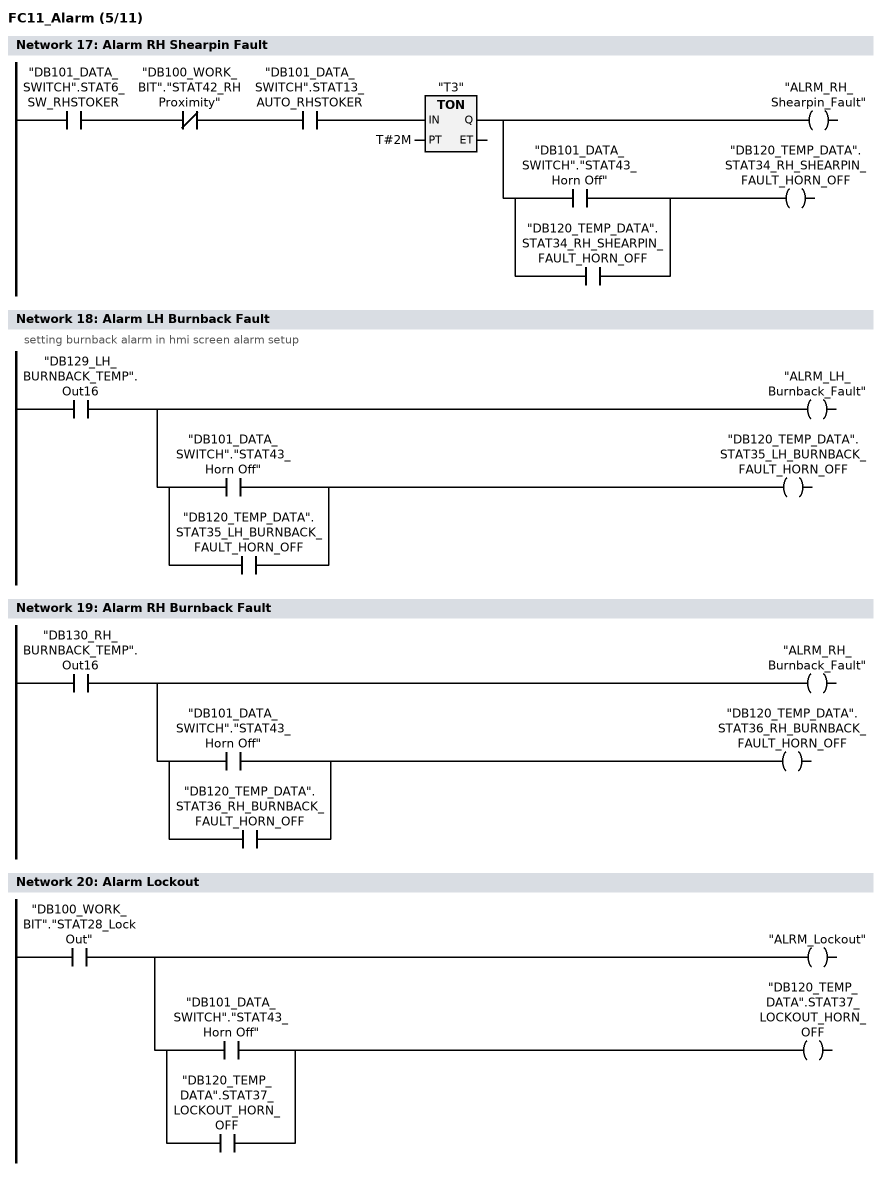
   "T3".TON(IN := "DB101_DATA_SWITCH".STAT6_SW_RHSTOKER AND NOT "DB100_WORK_BIT"."STAT42_RH Proximity" AND "DB101_DATA_SWITCH".STAT13_AUTO_RHSTOKER,
            PT := T#2M);
   "ALRM_RH_Shearpin_Fault" := "T3".Q;
   "DB120_TEMP_DATA".STAT34_RH_SHEARPIN_FAULT_HORN_OFF := "T3".Q AND ("DB101_DATA_SWITCH"."STAT43_Horn Off" OR "DB120_TEMP_DATA".STAT34_RH_SHEARPIN_FAULT_HORN_OFF);
END_REGION

REGION Network 18: Alarm LH Burnback Fault
   // setting burnback alarm in hmi screen alarm setup
   RUNG wire#powerrail
      Contact( "DB129_LH_BURNBACK_TEMP".Out16 )
      wire#w1
      Coil( "ALRM_LH_Burnback_Fault" )
   END_RUNG
   RUNG wire#w1
      Contact( "DB101_DATA_SWITCH"."STAT43_Horn Off" )
      wire#w2
      Coil( "DB120_TEMP_DATA".STAT35_LH_BURNBACK_FAULT_HORN_OFF )
   END_RUNG
   RUNG wire#w1
      Contact( "DB120_TEMP_DATA".STAT35_LH_BURNBACK_FAULT_HORN_OFF )
   END_RUNG wire#w2
   // the same network as SCL:
   "ALRM_LH_Burnback_Fault" := "DB129_LH_BURNBACK_TEMP".Out16;
   "DB120_TEMP_DATA".STAT35_LH_BURNBACK_FAULT_HORN_OFF := "DB129_LH_BURNBACK_TEMP".Out16 AND ("DB101_DATA_SWITCH"."STAT43_Horn Off" OR "DB120_TEMP_DATA".STAT35_LH_BURNBACK_FAULT_HORN_OFF);
END_REGION

REGION Network 19: Alarm RH Burnback Fault
   RUNG wire#powerrail
      Contact( "DB130_RH_BURNBACK_TEMP".Out16 )
      wire#w1
      Coil( "ALRM_RH_Burnback_Fault" )
   END_RUNG
   RUNG wire#w1
      Contact( "DB101_DATA_SWITCH"."STAT43_Horn Off" )
      wire#w2
      Coil( "DB120_TEMP_DATA".STAT36_RH_BURNBACK_FAULT_HORN_OFF )
   END_RUNG
   RUNG wire#w1
      Contact( "DB120_TEMP_DATA".STAT36_RH_BURNBACK_FAULT_HORN_OFF )
   END_RUNG wire#w2
   // the same network as SCL:
   "ALRM_RH_Burnback_Fault" := "DB130_RH_BURNBACK_TEMP".Out16;
   "DB120_TEMP_DATA".STAT36_RH_BURNBACK_FAULT_HORN_OFF := "DB130_RH_BURNBACK_TEMP".Out16 AND ("DB101_DATA_SWITCH"."STAT43_Horn Off" OR "DB120_TEMP_DATA".STAT36_RH_BURNBACK_FAULT_HORN_OFF);
END_REGION

REGION Network 20: Alarm Lockout
   RUNG wire#powerrail
      Contact( "DB100_WORK_BIT"."STAT28_Lock Out" )
      wire#w1
      Coil( "ALRM_Lockout" )
   END_RUNG
   RUNG wire#w1
      Contact( "DB101_DATA_SWITCH"."STAT43_Horn Off" )
      wire#w2
      Coil( "DB120_TEMP_DATA".STAT37_LOCKOUT_HORN_OFF )
   END_RUNG
   RUNG wire#w1
      Contact( "DB120_TEMP_DATA".STAT37_LOCKOUT_HORN_OFF )
   END_RUNG wire#w2
   // the same network as SCL:
   "ALRM_Lockout" := "DB100_WORK_BIT"."STAT28_Lock Out";
   "DB120_TEMP_DATA".STAT37_LOCKOUT_HORN_OFF := "DB100_WORK_BIT"."STAT28_Lock Out" AND ("DB101_DATA_SWITCH"."STAT43_Horn Off" OR "DB120_TEMP_DATA".STAT37_LOCKOUT_HORN_OFF);
END_REGION

REGION Network 21: Alarm Coal Hopper Low Level
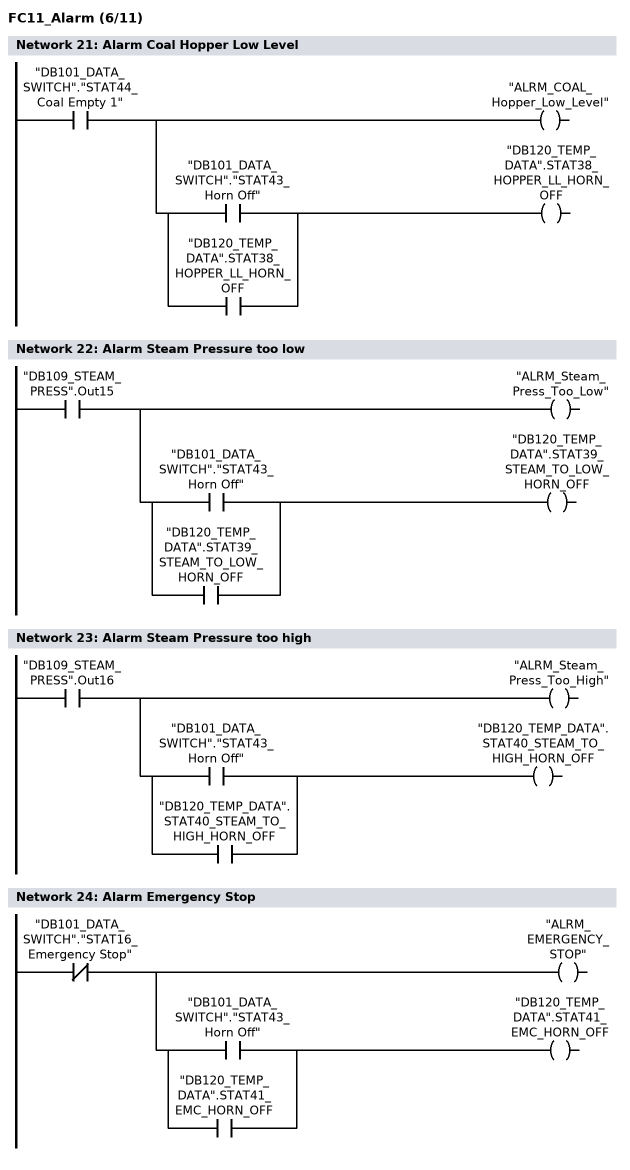
   RUNG wire#powerrail
      Contact( "DB101_DATA_SWITCH"."STAT44_Coal Empty 1" )
      wire#w1
      Coil( "ALRM_COAL_Hopper_Low_Level" )
   END_RUNG
   RUNG wire#w1
      Contact( "DB101_DATA_SWITCH"."STAT43_Horn Off" )
      wire#w2
      Coil( "DB120_TEMP_DATA".STAT38_HOPPER_LL_HORN_OFF )
   END_RUNG
   RUNG wire#w1
      Contact( "DB120_TEMP_DATA".STAT38_HOPPER_LL_HORN_OFF )
   END_RUNG wire#w2
   // the same network as SCL:
   "ALRM_COAL_Hopper_Low_Level" := "DB101_DATA_SWITCH"."STAT44_Coal Empty 1";
   "DB120_TEMP_DATA".STAT38_HOPPER_LL_HORN_OFF := "DB101_DATA_SWITCH"."STAT44_Coal Empty 1" AND ("DB101_DATA_SWITCH"."STAT43_Horn Off" OR "DB120_TEMP_DATA".STAT38_HOPPER_LL_HORN_OFF);
END_REGION

REGION Network 22: Alarm Steam Pressure too low
   RUNG wire#powerrail
      Contact( "DB109_STEAM_PRESS".Out15 )
      wire#w1
      Coil( "ALRM_Steam_Press_Too_Low" )
   END_RUNG
   RUNG wire#w1
      Contact( "DB101_DATA_SWITCH"."STAT43_Horn Off" )
      wire#w2
      Coil( "DB120_TEMP_DATA".STAT39_STEAM_TO_LOW_HORN_OFF )
   END_RUNG
   RUNG wire#w1
      Contact( "DB120_TEMP_DATA".STAT39_STEAM_TO_LOW_HORN_OFF )
   END_RUNG wire#w2
   // the same network as SCL:
   "ALRM_Steam_Press_Too_Low" := "DB109_STEAM_PRESS".Out15;
   "DB120_TEMP_DATA".STAT39_STEAM_TO_LOW_HORN_OFF := "DB109_STEAM_PRESS".Out15 AND ("DB101_DATA_SWITCH"."STAT43_Horn Off" OR "DB120_TEMP_DATA".STAT39_STEAM_TO_LOW_HORN_OFF);
END_REGION

REGION Network 23: Alarm Steam Pressure too high
   RUNG wire#powerrail
      Contact( "DB109_STEAM_PRESS".Out16 )
      wire#w1
      Coil( "ALRM_Steam_Press_Too_High" )
   END_RUNG
   RUNG wire#w1
      Contact( "DB101_DATA_SWITCH"."STAT43_Horn Off" )
      wire#w2
      Coil( "DB120_TEMP_DATA".STAT40_STEAM_TO_HIGH_HORN_OFF )
   END_RUNG
   RUNG wire#w1
      Contact( "DB120_TEMP_DATA".STAT40_STEAM_TO_HIGH_HORN_OFF )
   END_RUNG wire#w2
   // the same network as SCL:
   "ALRM_Steam_Press_Too_High" := "DB109_STEAM_PRESS".Out16;
   "DB120_TEMP_DATA".STAT40_STEAM_TO_HIGH_HORN_OFF := "DB109_STEAM_PRESS".Out16 AND ("DB101_DATA_SWITCH"."STAT43_Horn Off" OR "DB120_TEMP_DATA".STAT40_STEAM_TO_HIGH_HORN_OFF);
END_REGION

REGION Network 24: Alarm Emergency Stop
   RUNG wire#powerrail
      I_Contact( "DB101_DATA_SWITCH"."STAT16_Emergency Stop" )
      wire#w1
      Coil( "ALRM_EMERGENCY_STOP" )
   END_RUNG
   RUNG wire#w1
      Contact( "DB101_DATA_SWITCH"."STAT43_Horn Off" )
      wire#w2
      Coil( "DB120_TEMP_DATA".STAT41_EMC_HORN_OFF )
   END_RUNG
   RUNG wire#w1
      Contact( "DB120_TEMP_DATA".STAT41_EMC_HORN_OFF )
   END_RUNG wire#w2
   // the same network as SCL:
   "ALRM_EMERGENCY_STOP" := NOT "DB101_DATA_SWITCH"."STAT16_Emergency Stop";
   "DB120_TEMP_DATA".STAT41_EMC_HORN_OFF := NOT "DB101_DATA_SWITCH"."STAT16_Emergency Stop" AND ("DB101_DATA_SWITCH"."STAT43_Horn Off" OR "DB120_TEMP_DATA".STAT41_EMC_HORN_OFF);
END_REGION

REGION Network 25: Alarm Pump Pressure Low
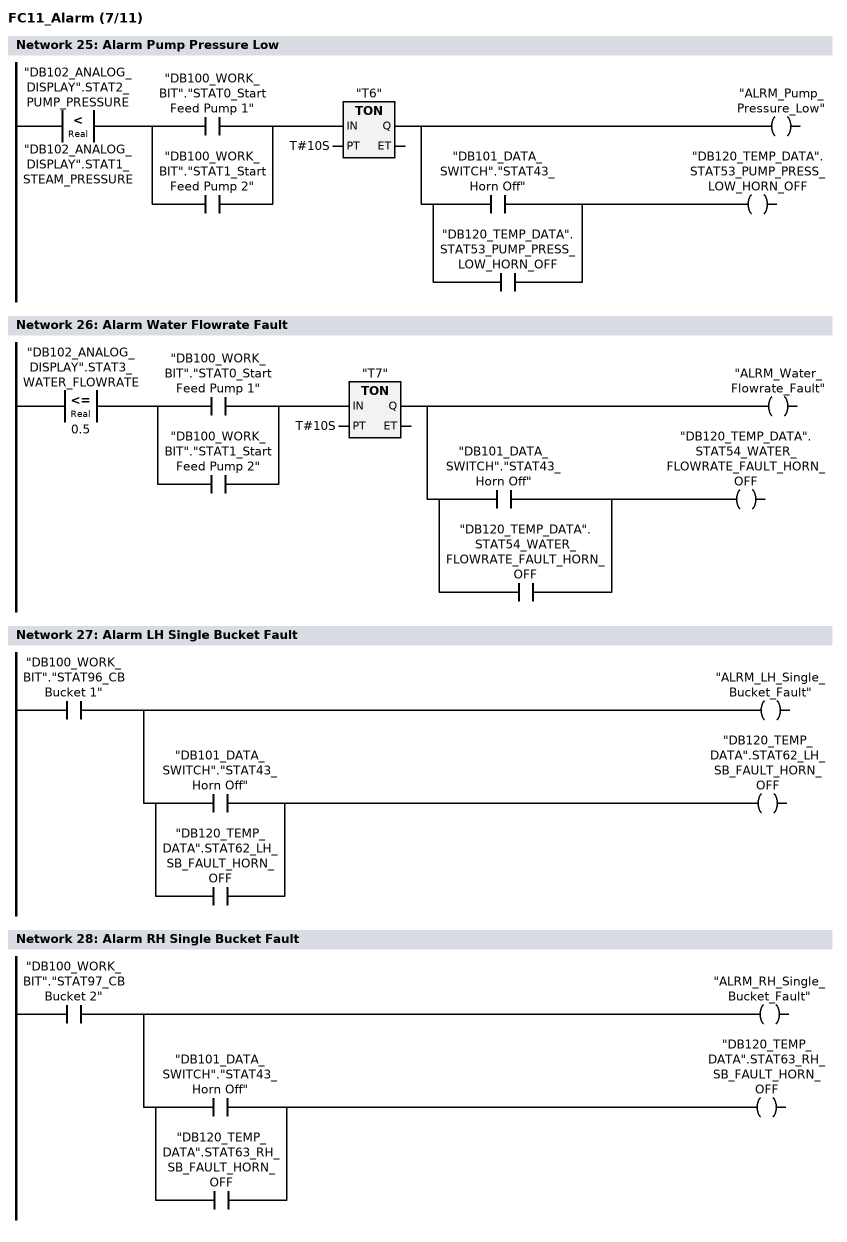
   "T6".TON(IN := ("DB102_ANALOG_DISPLAY".STAT2_PUMP_PRESSURE < "DB102_ANALOG_DISPLAY".STAT1_STEAM_PRESSURE) AND ("DB100_WORK_BIT"."STAT0_Start Feed Pump 1" OR "DB100_WORK_BIT"."STAT1_Start Feed Pump 2"),
            PT := T#10S);
   "ALRM_Pump_Pressure_Low" := "T6".Q;
   "DB120_TEMP_DATA".STAT53_PUMP_PRESS_LOW_HORN_OFF := "T6".Q AND ("DB101_DATA_SWITCH"."STAT43_Horn Off" OR "DB120_TEMP_DATA".STAT53_PUMP_PRESS_LOW_HORN_OFF);
END_REGION

REGION Network 26: Alarm Water Flowrate Fault
   "T7".TON(IN := ("DB102_ANALOG_DISPLAY".STAT3_WATER_FLOWRATE <= 0.5) AND ("DB100_WORK_BIT"."STAT0_Start Feed Pump 1" OR "DB100_WORK_BIT"."STAT1_Start Feed Pump 2"),
            PT := T#10S);
   "ALRM_Water_Flowrate_Fault" := "T7".Q;
   "DB120_TEMP_DATA".STAT54_WATER_FLOWRATE_FAULT_HORN_OFF := "T7".Q AND ("DB101_DATA_SWITCH"."STAT43_Horn Off" OR "DB120_TEMP_DATA".STAT54_WATER_FLOWRATE_FAULT_HORN_OFF);
END_REGION

REGION Network 27: Alarm LH Single Bucket Fault
   RUNG wire#powerrail
      Contact( "DB100_WORK_BIT"."STAT96_CB Bucket 1" )
      wire#w1
      Coil( "ALRM_LH_Single_Bucket_Fault" )
   END_RUNG
   RUNG wire#w1
      Contact( "DB101_DATA_SWITCH"."STAT43_Horn Off" )
      wire#w2
      Coil( "DB120_TEMP_DATA".STAT62_LH_SB_FAULT_HORN_OFF )
   END_RUNG
   RUNG wire#w1
      Contact( "DB120_TEMP_DATA".STAT62_LH_SB_FAULT_HORN_OFF )
   END_RUNG wire#w2
   // the same network as SCL:
   "ALRM_LH_Single_Bucket_Fault" := "DB100_WORK_BIT"."STAT96_CB Bucket 1";
   "DB120_TEMP_DATA".STAT62_LH_SB_FAULT_HORN_OFF := "DB100_WORK_BIT"."STAT96_CB Bucket 1" AND ("DB101_DATA_SWITCH"."STAT43_Horn Off" OR "DB120_TEMP_DATA".STAT62_LH_SB_FAULT_HORN_OFF);
END_REGION

REGION Network 28: Alarm RH Single Bucket Fault
   RUNG wire#powerrail
      Contact( "DB100_WORK_BIT"."STAT97_CB Bucket 2" )
      wire#w1
      Coil( "ALRM_RH_Single_Bucket_Fault" )
   END_RUNG
   RUNG wire#w1
      Contact( "DB101_DATA_SWITCH"."STAT43_Horn Off" )
      wire#w2
      Coil( "DB120_TEMP_DATA".STAT63_RH_SB_FAULT_HORN_OFF )
   END_RUNG
   RUNG wire#w1
      Contact( "DB120_TEMP_DATA".STAT63_RH_SB_FAULT_HORN_OFF )
   END_RUNG wire#w2
   // the same network as SCL:
   "ALRM_RH_Single_Bucket_Fault" := "DB100_WORK_BIT"."STAT97_CB Bucket 2";
   "DB120_TEMP_DATA".STAT63_RH_SB_FAULT_HORN_OFF := "DB100_WORK_BIT"."STAT97_CB Bucket 2" AND ("DB101_DATA_SWITCH"."STAT43_Horn Off" OR "DB120_TEMP_DATA".STAT63_RH_SB_FAULT_HORN_OFF);
END_REGION

REGION Network 29: Alarm FP Dry Run Protection
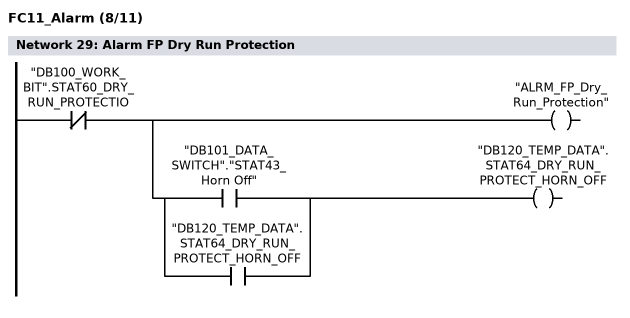
   RUNG wire#powerrail
      I_Contact( "DB100_WORK_BIT".STAT60_DRY_RUN_PROTECTIO )
      wire#w1
      Coil( "ALRM_FP_Dry_Run_Protection" )
   END_RUNG
   RUNG wire#w1
      Contact( "DB101_DATA_SWITCH"."STAT43_Horn Off" )
      wire#w2
      Coil( "DB120_TEMP_DATA".STAT64_DRY_RUN_PROTECT_HORN_OFF )
   END_RUNG
   RUNG wire#w1
      Contact( "DB120_TEMP_DATA".STAT64_DRY_RUN_PROTECT_HORN_OFF )
   END_RUNG wire#w2
   // the same network as SCL:
   "ALRM_FP_Dry_Run_Protection" := NOT "DB100_WORK_BIT".STAT60_DRY_RUN_PROTECTIO;
   "DB120_TEMP_DATA".STAT64_DRY_RUN_PROTECT_HORN_OFF := NOT "DB100_WORK_BIT".STAT60_DRY_RUN_PROTECTIO AND ("DB101_DATA_SWITCH"."STAT43_Horn Off" OR "DB120_TEMP_DATA".STAT64_DRY_RUN_PROTECT_HORN_OFF);
END_REGION

REGION Network 30: Alarm Horn
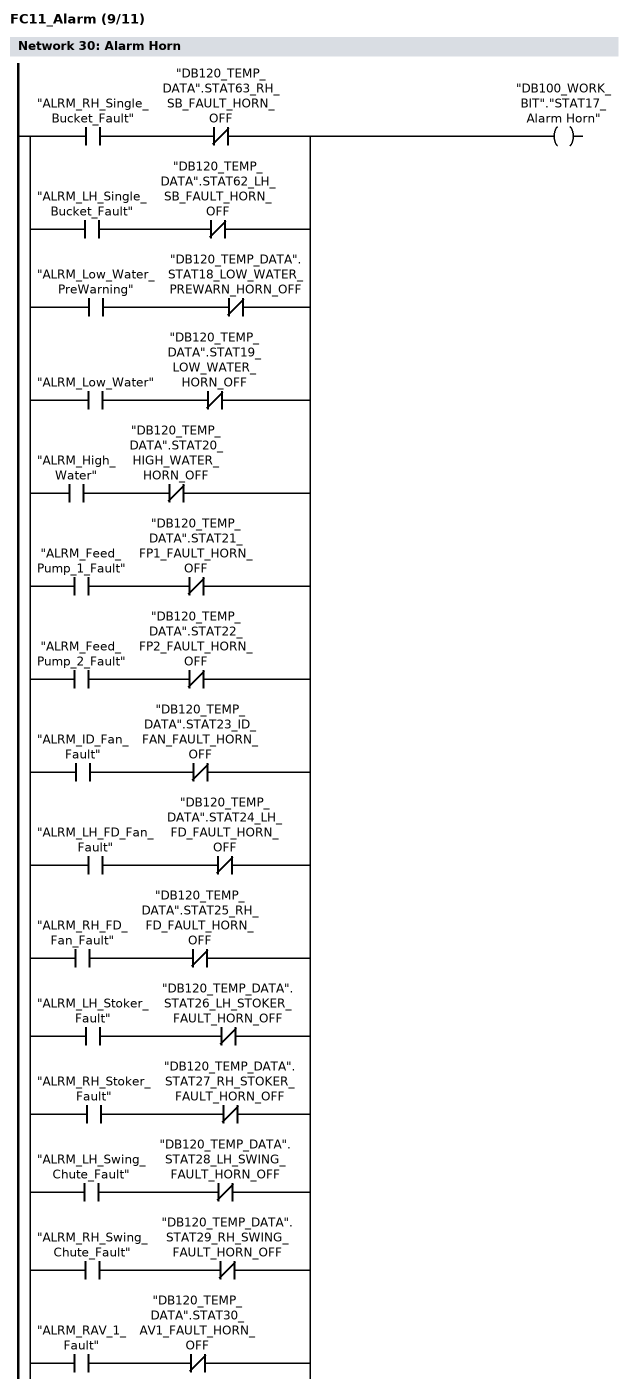
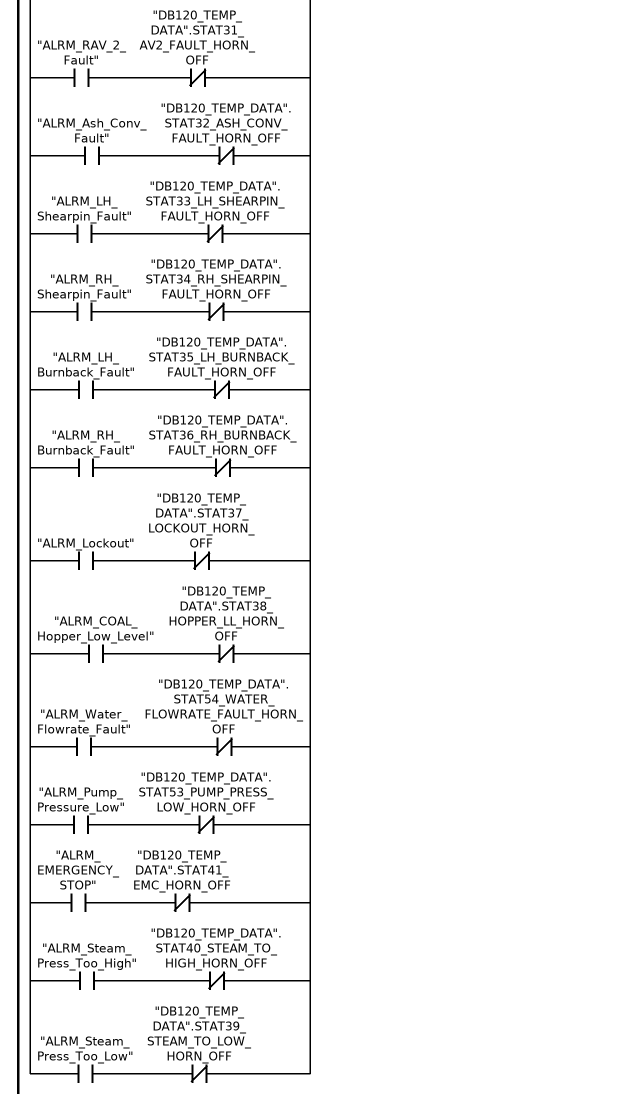
   RUNG wire#powerrail
      Contact( "ALRM_RH_Single_Bucket_Fault" )
      I_Contact( "DB120_TEMP_DATA".STAT63_RH_SB_FAULT_HORN_OFF )
      wire#w1
      Coil( "DB100_WORK_BIT"."STAT17_Alarm Horn" )
   END_RUNG
   RUNG wire#powerrail
      Contact( "ALRM_LH_Single_Bucket_Fault" )
      I_Contact( "DB120_TEMP_DATA".STAT62_LH_SB_FAULT_HORN_OFF )
   END_RUNG wire#w1
   RUNG wire#powerrail
      Contact( "ALRM_Low_Water_PreWarning" )
      I_Contact( "DB120_TEMP_DATA".STAT18_LOW_WATER_PREWARN_HORN_OFF )
   END_RUNG wire#w1
   RUNG wire#powerrail
      Contact( "ALRM_Low_Water" )
      I_Contact( "DB120_TEMP_DATA".STAT19_LOW_WATER_HORN_OFF )
   END_RUNG wire#w1
   RUNG wire#powerrail
      Contact( "ALRM_High_Water" )
      I_Contact( "DB120_TEMP_DATA".STAT20_HIGH_WATER_HORN_OFF )
   END_RUNG wire#w1
   RUNG wire#powerrail
      Contact( "ALRM_Feed_Pump_1_Fault" )
      I_Contact( "DB120_TEMP_DATA".STAT21_FP1_FAULT_HORN_OFF )
   END_RUNG wire#w1
   RUNG wire#powerrail
      Contact( "ALRM_Feed_Pump_2_Fault" )
      I_Contact( "DB120_TEMP_DATA".STAT22_FP2_FAULT_HORN_OFF )
   END_RUNG wire#w1
   RUNG wire#powerrail
      Contact( "ALRM_ID_Fan_Fault" )
      I_Contact( "DB120_TEMP_DATA".STAT23_ID_FAN_FAULT_HORN_OFF )
   END_RUNG wire#w1
   RUNG wire#powerrail
      Contact( "ALRM_LH_FD_Fan_Fault" )
      I_Contact( "DB120_TEMP_DATA".STAT24_LH_FD_FAULT_HORN_OFF )
   END_RUNG wire#w1
   RUNG wire#powerrail
      Contact( "ALRM_RH_FD_Fan_Fault" )
      I_Contact( "DB120_TEMP_DATA".STAT25_RH_FD_FAULT_HORN_OFF )
   END_RUNG wire#w1
   RUNG wire#powerrail
      Contact( "ALRM_LH_Stoker_Fault" )
      I_Contact( "DB120_TEMP_DATA".STAT26_LH_STOKER_FAULT_HORN_OFF )
   END_RUNG wire#w1
   RUNG wire#powerrail
      Contact( "ALRM_RH_Stoker_Fault" )
      I_Contact( "DB120_TEMP_DATA".STAT27_RH_STOKER_FAULT_HORN_OFF )
   END_RUNG wire#w1
   RUNG wire#powerrail
      Contact( "ALRM_LH_Swing_Chute_Fault" )
      I_Contact( "DB120_TEMP_DATA".STAT28_LH_SWING_FAULT_HORN_OFF )
   END_RUNG wire#w1
   RUNG wire#powerrail
      Contact( "ALRM_RH_Swing_Chute_Fault" )
      I_Contact( "DB120_TEMP_DATA".STAT29_RH_SWING_FAULT_HORN_OFF )
   END_RUNG wire#w1
   RUNG wire#powerrail
      Contact( "ALRM_RAV_1_Fault" )
      I_Contact( "DB120_TEMP_DATA".STAT30_AV1_FAULT_HORN_OFF )
   END_RUNG wire#w1
   RUNG wire#powerrail
      Contact( "ALRM_RAV_2_Fault" )
      I_Contact( "DB120_TEMP_DATA".STAT31_AV2_FAULT_HORN_OFF )
   END_RUNG wire#w1
   RUNG wire#powerrail
      Contact( "ALRM_Ash_Conv_Fault" )
      I_Contact( "DB120_TEMP_DATA".STAT32_ASH_CONV_FAULT_HORN_OFF )
   END_RUNG wire#w1
   RUNG wire#powerrail
      Contact( "ALRM_LH_Shearpin_Fault" )
      I_Contact( "DB120_TEMP_DATA".STAT33_LH_SHEARPIN_FAULT_HORN_OFF )
   END_RUNG wire#w1
   RUNG wire#powerrail
      Contact( "ALRM_RH_Shearpin_Fault" )
      I_Contact( "DB120_TEMP_DATA".STAT34_RH_SHEARPIN_FAULT_HORN_OFF )
   END_RUNG wire#w1
   RUNG wire#powerrail
      Contact( "ALRM_LH_Burnback_Fault" )
      I_Contact( "DB120_TEMP_DATA".STAT35_LH_BURNBACK_FAULT_HORN_OFF )
   END_RUNG wire#w1
   RUNG wire#powerrail
      Contact( "ALRM_RH_Burnback_Fault" )
      I_Contact( "DB120_TEMP_DATA".STAT36_RH_BURNBACK_FAULT_HORN_OFF )
   END_RUNG wire#w1
   RUNG wire#powerrail
      Contact( "ALRM_Lockout" )
      I_Contact( "DB120_TEMP_DATA".STAT37_LOCKOUT_HORN_OFF )
   END_RUNG wire#w1
   RUNG wire#powerrail
      Contact( "ALRM_COAL_Hopper_Low_Level" )
      I_Contact( "DB120_TEMP_DATA".STAT38_HOPPER_LL_HORN_OFF )
   END_RUNG wire#w1
   RUNG wire#powerrail
      Contact( "ALRM_Water_Flowrate_Fault" )
      I_Contact( "DB120_TEMP_DATA".STAT54_WATER_FLOWRATE_FAULT_HORN_OFF )
   END_RUNG wire#w1
   RUNG wire#powerrail
      Contact( "ALRM_Pump_Pressure_Low" )
      I_Contact( "DB120_TEMP_DATA".STAT53_PUMP_PRESS_LOW_HORN_OFF )
   END_RUNG wire#w1
   RUNG wire#powerrail
      Contact( "ALRM_EMERGENCY_STOP" )
      I_Contact( "DB120_TEMP_DATA".STAT41_EMC_HORN_OFF )
   END_RUNG wire#w1
   RUNG wire#powerrail
      Contact( "ALRM_Steam_Press_Too_High" )
      I_Contact( "DB120_TEMP_DATA".STAT40_STEAM_TO_HIGH_HORN_OFF )
   END_RUNG wire#w1
   RUNG wire#powerrail
      Contact( "ALRM_Steam_Press_Too_Low" )
      I_Contact( "DB120_TEMP_DATA".STAT39_STEAM_TO_LOW_HORN_OFF )
   END_RUNG wire#w1
   // the same network as SCL:
   "DB100_WORK_BIT"."STAT17_Alarm Horn" := ("ALRM_RH_Single_Bucket_Fault" AND NOT "DB120_TEMP_DATA".STAT63_RH_SB_FAULT_HORN_OFF) OR ("ALRM_LH_Single_Bucket_Fault" AND NOT "DB120_TEMP_DATA".STAT62_LH_SB_FAULT_HORN_OFF) OR ("ALRM_Low_Water_PreWarning" AND NOT "DB120_TEMP_DATA".STAT18_LOW_WATER_PREWARN_HORN_OFF) OR ("ALRM_Low_Water" AND NOT "DB120_TEMP_DATA".STAT19_LOW_WATER_HORN_OFF) OR ("ALRM_High_Water" AND NOT "DB120_TEMP_DATA".STAT20_HIGH_WATER_HORN_OFF) OR ("ALRM_Feed_Pump_1_Fault" AND NOT "DB120_TEMP_DATA".STAT21_FP1_FAULT_HORN_OFF) OR ("ALRM_Feed_Pump_2_Fault" AND NOT "DB120_TEMP_DATA".STAT22_FP2_FAULT_HORN_OFF) OR ("ALRM_ID_Fan_Fault" AND NOT "DB120_TEMP_DATA".STAT23_ID_FAN_FAULT_HORN_OFF) OR ("ALRM_LH_FD_Fan_Fault" AND NOT "DB120_TEMP_DATA".STAT24_LH_FD_FAULT_HORN_OFF) OR ("ALRM_RH_FD_Fan_Fault" AND NOT "DB120_TEMP_DATA".STAT25_RH_FD_FAULT_HORN_OFF) OR ("ALRM_LH_Stoker_Fault" AND NOT "DB120_TEMP_DATA".STAT26_LH_STOKER_FAULT_HORN_OFF) OR ("ALRM_RH_Stoker_Fault" AND NOT "DB120_TEMP_DATA".STAT27_RH_STOKER_FAULT_HORN_OFF) OR ("ALRM_LH_Swing_Chute_Fault" AND NOT "DB120_TEMP_DATA".STAT28_LH_SWING_FAULT_HORN_OFF) OR ("ALRM_RH_Swing_Chute_Fault" AND NOT "DB120_TEMP_DATA".STAT29_RH_SWING_FAULT_HORN_OFF) OR ("ALRM_RAV_1_Fault" AND NOT "DB120_TEMP_DATA".STAT30_AV1_FAULT_HORN_OFF) OR ("ALRM_RAV_2_Fault" AND NOT "DB120_TEMP_DATA".STAT31_AV2_FAULT_HORN_OFF) OR ("ALRM_Ash_Conv_Fault" AND NOT "DB120_TEMP_DATA".STAT32_ASH_CONV_FAULT_HORN_OFF) OR ("ALRM_LH_Shearpin_Fault" AND NOT "DB120_TEMP_DATA".STAT33_LH_SHEARPIN_FAULT_HORN_OFF) OR ("ALRM_RH_Shearpin_Fault" AND NOT "DB120_TEMP_DATA".STAT34_RH_SHEARPIN_FAULT_HORN_OFF) OR ("ALRM_LH_Burnback_Fault" AND NOT "DB120_TEMP_DATA".STAT35_LH_BURNBACK_FAULT_HORN_OFF) OR ("ALRM_RH_Burnback_Fault" AND NOT "DB120_TEMP_DATA".STAT36_RH_BURNBACK_FAULT_HORN_OFF) OR ("ALRM_Lockout" AND NOT "DB120_TEMP_DATA".STAT37_LOCKOUT_HORN_OFF) OR ("ALRM_COAL_Hopper_Low_Level" AND NOT "DB120_TEMP_DATA".STAT38_HOPPER_LL_HORN_OFF) OR ("ALRM_Water_Flowrate_Fault" AND NOT "DB120_TEMP_DATA".STAT54_WATER_FLOWRATE_FAULT_HORN_OFF) OR ("ALRM_Pump_Pressure_Low" AND NOT "DB120_TEMP_DATA".STAT53_PUMP_PRESS_LOW_HORN_OFF) OR ("ALRM_EMERGENCY_STOP" AND NOT "DB120_TEMP_DATA".STAT41_EMC_HORN_OFF) OR ("ALRM_Steam_Press_Too_High" AND NOT "DB120_TEMP_DATA".STAT40_STEAM_TO_HIGH_HORN_OFF) OR ("ALRM_Steam_Press_Too_Low" AND NOT "DB120_TEMP_DATA".STAT39_STEAM_TO_LOW_HORN_OFF);
END_REGION

REGION Network 31: STL Network 31 Alarm Flash COMMAND | CHANGEOVER HORN OFF SWITCH | I 5.6
   // if switch horn of change then alarm flash command set
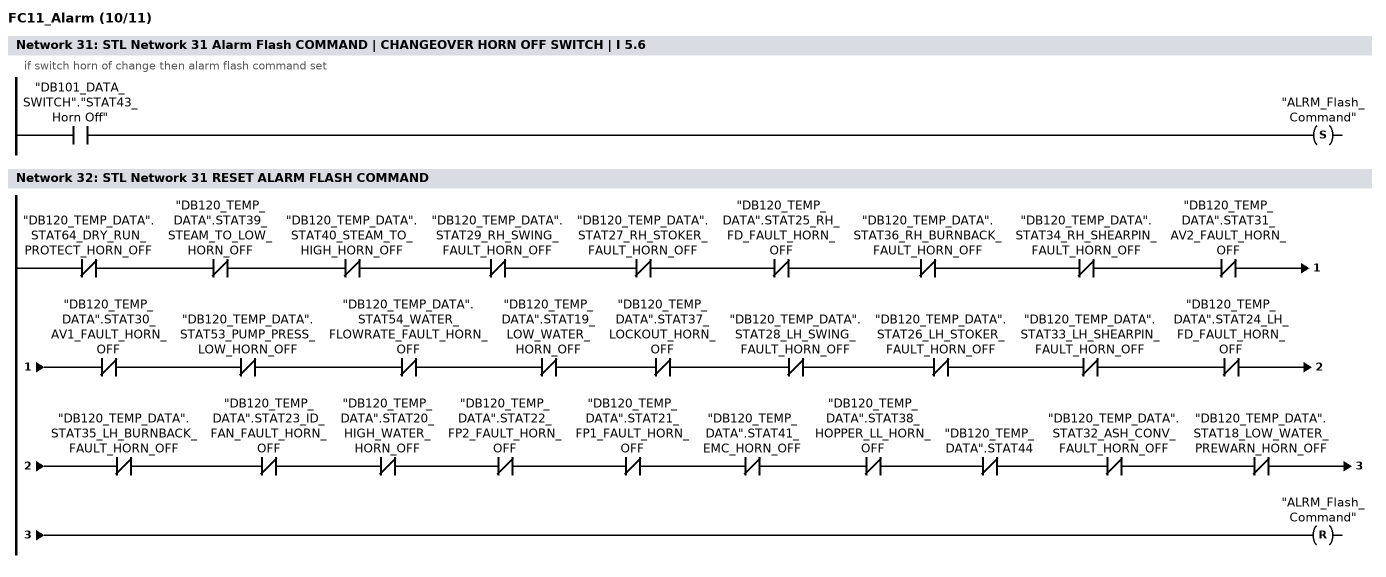
   RUNG wire#powerrail
      Contact( "DB101_DATA_SWITCH"."STAT43_Horn Off" )
      S_Coil( "ALRM_Flash_Command" )
   END_RUNG
   // the same network as SCL:
   IF "DB101_DATA_SWITCH"."STAT43_Horn Off" THEN "ALRM_Flash_Command" := TRUE; END_IF;
END_REGION

REGION Network 32: STL Network 31 RESET ALARM FLASH COMMAND
   RUNG wire#powerrail
      I_Contact( "DB120_TEMP_DATA".STAT64_DRY_RUN_PROTECT_HORN_OFF )
      I_Contact( "DB120_TEMP_DATA".STAT39_STEAM_TO_LOW_HORN_OFF )
      I_Contact( "DB120_TEMP_DATA".STAT40_STEAM_TO_HIGH_HORN_OFF )
      I_Contact( "DB120_TEMP_DATA".STAT29_RH_SWING_FAULT_HORN_OFF )
      I_Contact( "DB120_TEMP_DATA".STAT27_RH_STOKER_FAULT_HORN_OFF )
      I_Contact( "DB120_TEMP_DATA".STAT25_RH_FD_FAULT_HORN_OFF )
      I_Contact( "DB120_TEMP_DATA".STAT36_RH_BURNBACK_FAULT_HORN_OFF )
      I_Contact( "DB120_TEMP_DATA".STAT34_RH_SHEARPIN_FAULT_HORN_OFF )
      I_Contact( "DB120_TEMP_DATA".STAT31_AV2_FAULT_HORN_OFF )
      I_Contact( "DB120_TEMP_DATA".STAT30_AV1_FAULT_HORN_OFF )
      I_Contact( "DB120_TEMP_DATA".STAT53_PUMP_PRESS_LOW_HORN_OFF )
      I_Contact( "DB120_TEMP_DATA".STAT54_WATER_FLOWRATE_FAULT_HORN_OFF )
      I_Contact( "DB120_TEMP_DATA".STAT19_LOW_WATER_HORN_OFF )
      I_Contact( "DB120_TEMP_DATA".STAT37_LOCKOUT_HORN_OFF )
      I_Contact( "DB120_TEMP_DATA".STAT28_LH_SWING_FAULT_HORN_OFF )
      I_Contact( "DB120_TEMP_DATA".STAT26_LH_STOKER_FAULT_HORN_OFF )
      I_Contact( "DB120_TEMP_DATA".STAT33_LH_SHEARPIN_FAULT_HORN_OFF )
      I_Contact( "DB120_TEMP_DATA".STAT24_LH_FD_FAULT_HORN_OFF )
      I_Contact( "DB120_TEMP_DATA".STAT35_LH_BURNBACK_FAULT_HORN_OFF )
      I_Contact( "DB120_TEMP_DATA".STAT23_ID_FAN_FAULT_HORN_OFF )
      I_Contact( "DB120_TEMP_DATA".STAT20_HIGH_WATER_HORN_OFF )
      I_Contact( "DB120_TEMP_DATA".STAT22_FP2_FAULT_HORN_OFF )
      I_Contact( "DB120_TEMP_DATA".STAT21_FP1_FAULT_HORN_OFF )
      I_Contact( "DB120_TEMP_DATA".STAT41_EMC_HORN_OFF )
      I_Contact( "DB120_TEMP_DATA".STAT38_HOPPER_LL_HORN_OFF )
      I_Contact( "DB120_TEMP_DATA".STAT44 )
      I_Contact( "DB120_TEMP_DATA".STAT32_ASH_CONV_FAULT_HORN_OFF )
      I_Contact( "DB120_TEMP_DATA".STAT18_LOW_WATER_PREWARN_HORN_OFF )
      R_Coil( "ALRM_Flash_Command" )
   END_RUNG
   // the same network as SCL:
   IF NOT "DB120_TEMP_DATA".STAT64_DRY_RUN_PROTECT_HORN_OFF AND NOT "DB120_TEMP_DATA".STAT39_STEAM_TO_LOW_HORN_OFF AND NOT "DB120_TEMP_DATA".STAT40_STEAM_TO_HIGH_HORN_OFF AND NOT "DB120_TEMP_DATA".STAT29_RH_SWING_FAULT_HORN_OFF AND NOT "DB120_TEMP_DATA".STAT27_RH_STOKER_FAULT_HORN_OFF AND NOT "DB120_TEMP_DATA".STAT25_RH_FD_FAULT_HORN_OFF AND NOT "DB120_TEMP_DATA".STAT36_RH_BURNBACK_FAULT_HORN_OFF AND NOT "DB120_TEMP_DATA".STAT34_RH_SHEARPIN_FAULT_HORN_OFF AND NOT "DB120_TEMP_DATA".STAT31_AV2_FAULT_HORN_OFF AND NOT "DB120_TEMP_DATA".STAT30_AV1_FAULT_HORN_OFF AND NOT "DB120_TEMP_DATA".STAT53_PUMP_PRESS_LOW_HORN_OFF AND NOT "DB120_TEMP_DATA".STAT54_WATER_FLOWRATE_FAULT_HORN_OFF AND NOT "DB120_TEMP_DATA".STAT19_LOW_WATER_HORN_OFF AND NOT "DB120_TEMP_DATA".STAT37_LOCKOUT_HORN_OFF AND NOT "DB120_TEMP_DATA".STAT28_LH_SWING_FAULT_HORN_OFF AND NOT "DB120_TEMP_DATA".STAT26_LH_STOKER_FAULT_HORN_OFF AND NOT "DB120_TEMP_DATA".STAT33_LH_SHEARPIN_FAULT_HORN_OFF AND NOT "DB120_TEMP_DATA".STAT24_LH_FD_FAULT_HORN_OFF AND NOT "DB120_TEMP_DATA".STAT35_LH_BURNBACK_FAULT_HORN_OFF AND NOT "DB120_TEMP_DATA".STAT23_ID_FAN_FAULT_HORN_OFF AND NOT "DB120_TEMP_DATA".STAT20_HIGH_WATER_HORN_OFF AND NOT "DB120_TEMP_DATA".STAT22_FP2_FAULT_HORN_OFF AND NOT "DB120_TEMP_DATA".STAT21_FP1_FAULT_HORN_OFF AND NOT "DB120_TEMP_DATA".STAT41_EMC_HORN_OFF AND NOT "DB120_TEMP_DATA".STAT38_HOPPER_LL_HORN_OFF AND NOT "DB120_TEMP_DATA".STAT44 AND NOT "DB120_TEMP_DATA".STAT32_ASH_CONV_FAULT_HORN_OFF AND NOT "DB120_TEMP_DATA".STAT18_LOW_WATER_PREWARN_HORN_OFF THEN
       "ALRM_Flash_Command" := FALSE;
   END_IF;
END_REGION

REGION Network 33: STL Network 31
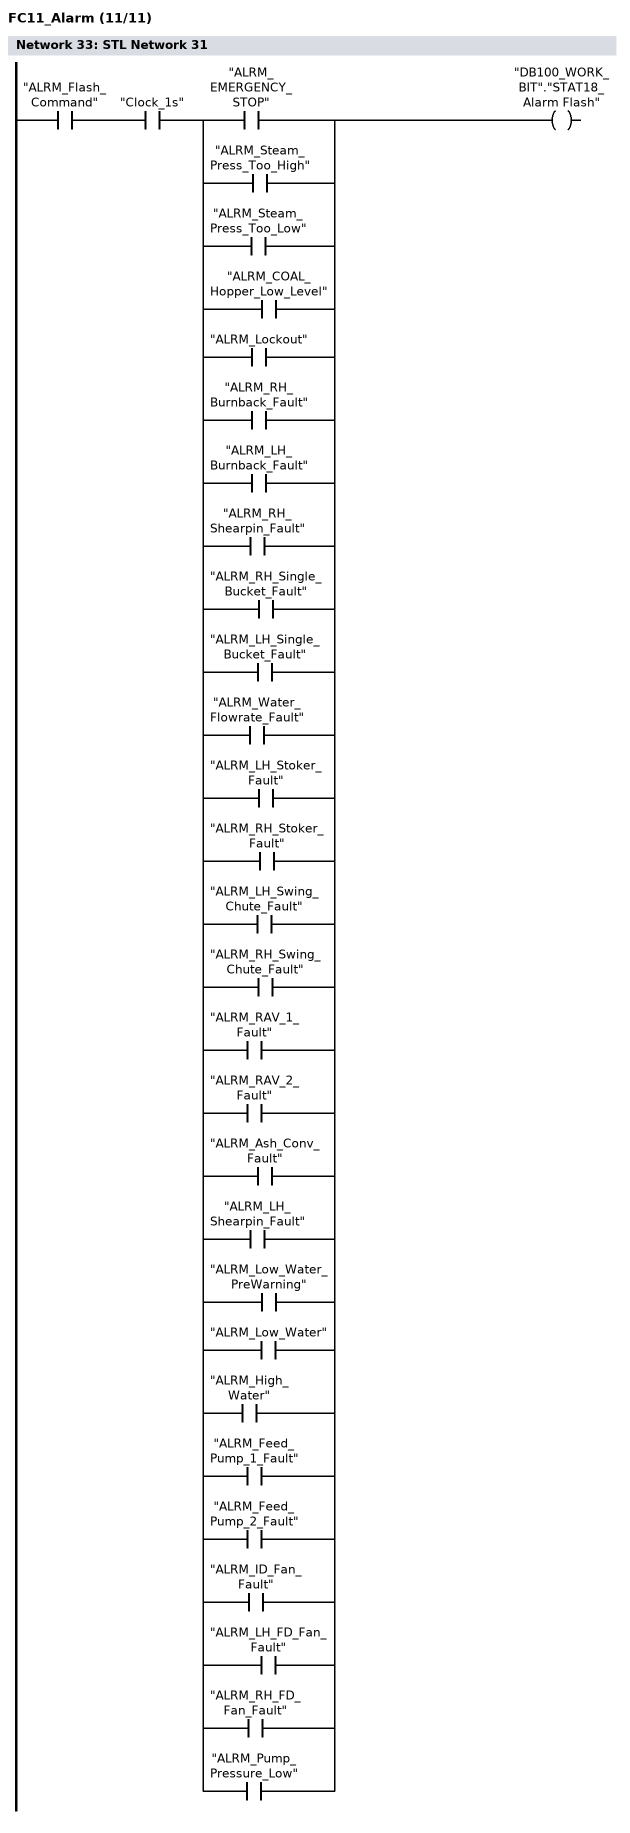
   RUNG wire#powerrail
      Contact( "ALRM_Flash_Command" )
      Contact( "Clock_1s" )
      wire#w1
      Contact( "ALRM_EMERGENCY_STOP" )
      wire#w2
      Coil( "DB100_WORK_BIT"."STAT18_Alarm Flash" )
   END_RUNG
   RUNG wire#w1
      Contact( "ALRM_Steam_Press_Too_High" )
   END_RUNG wire#w2
   RUNG wire#w1
      Contact( "ALRM_Steam_Press_Too_Low" )
   END_RUNG wire#w2
   RUNG wire#w1
      Contact( "ALRM_COAL_Hopper_Low_Level" )
   END_RUNG wire#w2
   RUNG wire#w1
      Contact( "ALRM_Lockout" )
   END_RUNG wire#w2
   RUNG wire#w1
      Contact( "ALRM_RH_Burnback_Fault" )
   END_RUNG wire#w2
   RUNG wire#w1
      Contact( "ALRM_LH_Burnback_Fault" )
   END_RUNG wire#w2
   RUNG wire#w1
      Contact( "ALRM_RH_Shearpin_Fault" )
   END_RUNG wire#w2
   RUNG wire#w1
      Contact( "ALRM_RH_Single_Bucket_Fault" )
   END_RUNG wire#w2
   RUNG wire#w1
      Contact( "ALRM_LH_Single_Bucket_Fault" )
   END_RUNG wire#w2
   RUNG wire#w1
      Contact( "ALRM_Water_Flowrate_Fault" )
   END_RUNG wire#w2
   RUNG wire#w1
      Contact( "ALRM_LH_Stoker_Fault" )
   END_RUNG wire#w2
   RUNG wire#w1
      Contact( "ALRM_RH_Stoker_Fault" )
   END_RUNG wire#w2
   RUNG wire#w1
      Contact( "ALRM_LH_Swing_Chute_Fault" )
   END_RUNG wire#w2
   RUNG wire#w1
      Contact( "ALRM_RH_Swing_Chute_Fault" )
   END_RUNG wire#w2
   RUNG wire#w1
      Contact( "ALRM_RAV_1_Fault" )
   END_RUNG wire#w2
   RUNG wire#w1
      Contact( "ALRM_RAV_2_Fault" )
   END_RUNG wire#w2
   RUNG wire#w1
      Contact( "ALRM_Ash_Conv_Fault" )
   END_RUNG wire#w2
   RUNG wire#w1
      Contact( "ALRM_LH_Shearpin_Fault" )
   END_RUNG wire#w2
   RUNG wire#w1
      Contact( "ALRM_Low_Water_PreWarning" )
   END_RUNG wire#w2
   RUNG wire#w1
      Contact( "ALRM_Low_Water" )
   END_RUNG wire#w2
   RUNG wire#w1
      Contact( "ALRM_High_Water" )
   END_RUNG wire#w2
   RUNG wire#w1
      Contact( "ALRM_Feed_Pump_1_Fault" )
   END_RUNG wire#w2
   RUNG wire#w1
      Contact( "ALRM_Feed_Pump_2_Fault" )
   END_RUNG wire#w2
   RUNG wire#w1
      Contact( "ALRM_ID_Fan_Fault" )
   END_RUNG wire#w2
   RUNG wire#w1
      Contact( "ALRM_LH_FD_Fan_Fault" )
   END_RUNG wire#w2
   RUNG wire#w1
      Contact( "ALRM_RH_FD_Fan_Fault" )
   END_RUNG wire#w2
   RUNG wire#w1
      Contact( "ALRM_Pump_Pressure_Low" )
   END_RUNG wire#w2
   // the same network as SCL:
   "DB100_WORK_BIT"."STAT18_Alarm Flash" := "ALRM_Flash_Command" AND "Clock_1s" AND ("ALRM_EMERGENCY_STOP" OR "ALRM_Steam_Press_Too_High" OR "ALRM_Steam_Press_Too_Low" OR "ALRM_COAL_Hopper_Low_Level" OR "ALRM_Lockout" OR "ALRM_RH_Burnback_Fault" OR "ALRM_LH_Burnback_Fault" OR "ALRM_RH_Shearpin_Fault" OR "ALRM_RH_Single_Bucket_Fault" OR "ALRM_LH_Single_Bucket_Fault" OR "ALRM_Water_Flowrate_Fault" OR "ALRM_LH_Stoker_Fault" OR "ALRM_RH_Stoker_Fault" OR "ALRM_LH_Swing_Chute_Fault" OR "ALRM_RH_Swing_Chute_Fault" OR "ALRM_RAV_1_Fault" OR "ALRM_RAV_2_Fault" OR "ALRM_Ash_Conv_Fault" OR "ALRM_LH_Shearpin_Fault" OR "ALRM_Low_Water_PreWarning" OR "ALRM_Low_Water" OR "ALRM_High_Water" OR "ALRM_Feed_Pump_1_Fault" OR "ALRM_Feed_Pump_2_Fault" OR "ALRM_ID_Fan_Fault" OR "ALRM_LH_FD_Fan_Fault" OR "ALRM_RH_FD_Fan_Fault" OR "ALRM_Pump_Pressure_Low");
END_REGION
END_FUNCTION

FUNCTION "FC15_Digital_Input" : Void   // FC15, LAD
TITLE = Mapping Digital Input to DB 101
{ S7_Optimized_Access := 'TRUE' }
VERSION : 0.1
BEGIN

REGION Network 1: EMERGENCY STOP (I0.0)
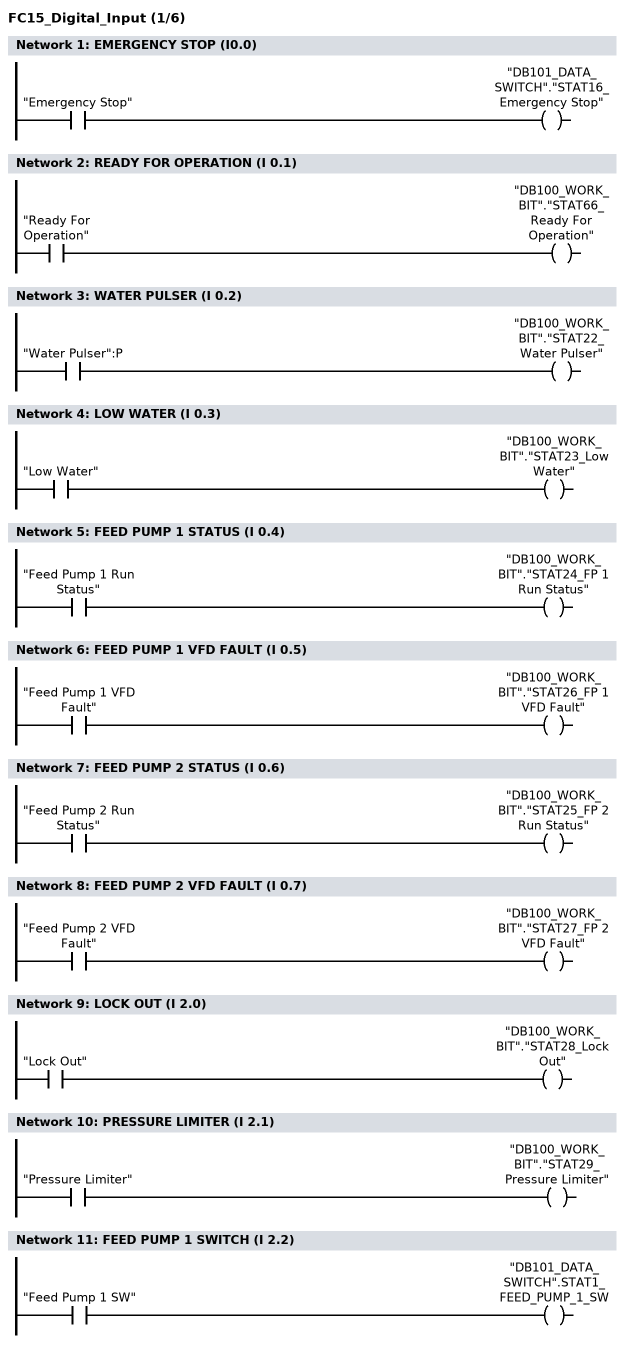
   RUNG wire#powerrail
      Contact( "Emergency Stop" )
      Coil( "DB101_DATA_SWITCH"."STAT16_Emergency Stop" )
   END_RUNG
   // the same network as SCL:
   "DB101_DATA_SWITCH"."STAT16_Emergency Stop" := "Emergency Stop";
END_REGION

REGION Network 2: READY FOR OPERATION (I 0.1)
   RUNG wire#powerrail
      Contact( "Ready For Operation" )
      Coil( "DB100_WORK_BIT"."STAT66_Ready For Operation" )
   END_RUNG
   // the same network as SCL:
   "DB100_WORK_BIT"."STAT66_Ready For Operation" := "Ready For Operation";
END_REGION

REGION Network 3: WATER PULSER (I 0.2)
   RUNG wire#powerrail
      Contact( "Water Pulser":P )
      Coil( "DB100_WORK_BIT"."STAT22_Water Pulser" )
   END_RUNG
   // the same network as SCL:
   "DB100_WORK_BIT"."STAT22_Water Pulser" := "Water Pulser":P;
END_REGION

REGION Network 4: LOW WATER (I 0.3)
   RUNG wire#powerrail
      Contact( "Low Water" )
      Coil( "DB100_WORK_BIT"."STAT23_Low Water" )
   END_RUNG
   // the same network as SCL:
   "DB100_WORK_BIT"."STAT23_Low Water" := "Low Water";
END_REGION

REGION Network 5: FEED PUMP 1 STATUS (I 0.4)
   RUNG wire#powerrail
      Contact( "Feed Pump 1 Run Status" )
      Coil( "DB100_WORK_BIT"."STAT24_FP 1 Run Status" )
   END_RUNG
   // the same network as SCL:
   "DB100_WORK_BIT"."STAT24_FP 1 Run Status" := "Feed Pump 1 Run Status";
END_REGION

REGION Network 6: FEED PUMP 1 VFD FAULT (I 0.5)
   RUNG wire#powerrail
      Contact( "Feed Pump 1 VFD Fault" )
      Coil( "DB100_WORK_BIT"."STAT26_FP 1 VFD Fault" )
   END_RUNG
   // the same network as SCL:
   "DB100_WORK_BIT"."STAT26_FP 1 VFD Fault" := "Feed Pump 1 VFD Fault";
END_REGION

REGION Network 7: FEED PUMP 2 STATUS (I 0.6)
   RUNG wire#powerrail
      Contact( "Feed Pump 2 Run Status" )
      Coil( "DB100_WORK_BIT"."STAT25_FP 2 Run Status" )
   END_RUNG
   // the same network as SCL:
   "DB100_WORK_BIT"."STAT25_FP 2 Run Status" := "Feed Pump 2 Run Status";
END_REGION

REGION Network 8: FEED PUMP 2 VFD FAULT (I 0.7)
   RUNG wire#powerrail
      Contact( "Feed Pump 2 VFD Fault" )
      Coil( "DB100_WORK_BIT"."STAT27_FP 2 VFD Fault" )
   END_RUNG
   // the same network as SCL:
   "DB100_WORK_BIT"."STAT27_FP 2 VFD Fault" := "Feed Pump 2 VFD Fault";
END_REGION

REGION Network 9: LOCK OUT (I 2.0)
   RUNG wire#powerrail
      Contact( "Lock Out" )
      Coil( "DB100_WORK_BIT"."STAT28_Lock Out" )
   END_RUNG
   // the same network as SCL:
   "DB100_WORK_BIT"."STAT28_Lock Out" := "Lock Out";
END_REGION

REGION Network 10: PRESSURE LIMITER (I 2.1)
   RUNG wire#powerrail
      Contact( "Pressure Limiter" )
      Coil( "DB100_WORK_BIT"."STAT29_Pressure Limiter" )
   END_RUNG
   // the same network as SCL:
   "DB100_WORK_BIT"."STAT29_Pressure Limiter" := "Pressure Limiter";
END_REGION

REGION Network 11: FEED PUMP 1 SWITCH (I 2.2)
   RUNG wire#powerrail
      Contact( "Feed Pump 1 SW" )
      Coil( "DB101_DATA_SWITCH".STAT1_FEED_PUMP_1_SW )
   END_RUNG
   // the same network as SCL:
   "DB101_DATA_SWITCH".STAT1_FEED_PUMP_1_SW := "Feed Pump 1 SW";
END_REGION

REGION Network 12: FEED PUMP 2 SWITCH (I 2.3)
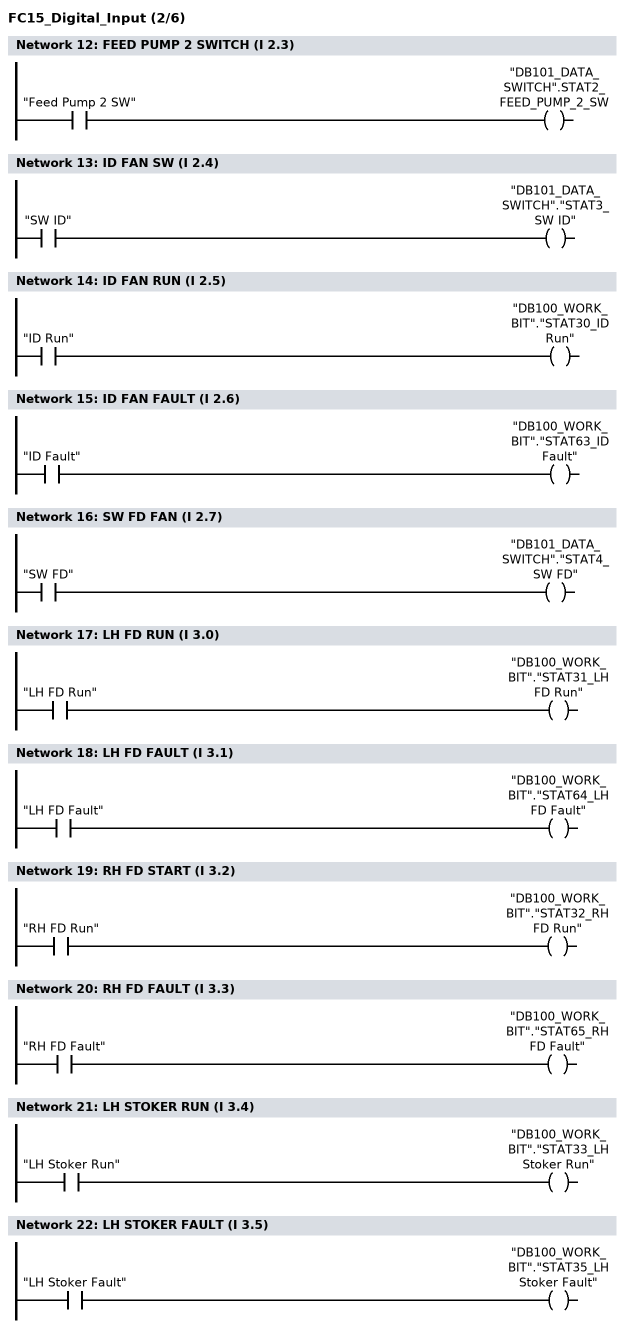
   RUNG wire#powerrail
      Contact( "Feed Pump 2 SW" )
      Coil( "DB101_DATA_SWITCH".STAT2_FEED_PUMP_2_SW )
   END_RUNG
   // the same network as SCL:
   "DB101_DATA_SWITCH".STAT2_FEED_PUMP_2_SW := "Feed Pump 2 SW";
END_REGION

REGION Network 13: ID FAN SW (I 2.4)
   RUNG wire#powerrail
      Contact( "SW ID" )
      Coil( "DB101_DATA_SWITCH"."STAT3_SW ID" )
   END_RUNG
   // the same network as SCL:
   "DB101_DATA_SWITCH"."STAT3_SW ID" := "SW ID";
END_REGION

REGION Network 14: ID FAN RUN (I 2.5)
   RUNG wire#powerrail
      Contact( "ID Run" )
      Coil( "DB100_WORK_BIT"."STAT30_ID Run" )
   END_RUNG
   // the same network as SCL:
   "DB100_WORK_BIT"."STAT30_ID Run" := "ID Run";
END_REGION

REGION Network 15: ID FAN FAULT (I 2.6)
   RUNG wire#powerrail
      Contact( "ID Fault" )
      Coil( "DB100_WORK_BIT"."STAT63_ID Fault" )
   END_RUNG
   // the same network as SCL:
   "DB100_WORK_BIT"."STAT63_ID Fault" := "ID Fault";
END_REGION

REGION Network 16: SW FD FAN (I 2.7)
   RUNG wire#powerrail
      Contact( "SW FD" )
      Coil( "DB101_DATA_SWITCH"."STAT4_SW FD" )
   END_RUNG
   // the same network as SCL:
   "DB101_DATA_SWITCH"."STAT4_SW FD" := "SW FD";
END_REGION

REGION Network 17: LH FD RUN (I 3.0)
   RUNG wire#powerrail
      Contact( "LH FD Run" )
      Coil( "DB100_WORK_BIT"."STAT31_LH FD Run" )
   END_RUNG
   // the same network as SCL:
   "DB100_WORK_BIT"."STAT31_LH FD Run" := "LH FD Run";
END_REGION

REGION Network 18: LH FD FAULT (I 3.1)
   RUNG wire#powerrail
      Contact( "LH FD Fault" )
      Coil( "DB100_WORK_BIT"."STAT64_LH FD Fault" )
   END_RUNG
   // the same network as SCL:
   "DB100_WORK_BIT"."STAT64_LH FD Fault" := "LH FD Fault";
END_REGION

REGION Network 19: RH FD START (I 3.2)
   RUNG wire#powerrail
      Contact( "RH FD Run" )
      Coil( "DB100_WORK_BIT"."STAT32_RH FD Run" )
   END_RUNG
   // the same network as SCL:
   "DB100_WORK_BIT"."STAT32_RH FD Run" := "RH FD Run";
END_REGION

REGION Network 20: RH FD FAULT (I 3.3)
   RUNG wire#powerrail
      Contact( "RH FD Fault" )
      Coil( "DB100_WORK_BIT"."STAT65_RH FD Fault" )
   END_RUNG
   // the same network as SCL:
   "DB100_WORK_BIT"."STAT65_RH FD Fault" := "RH FD Fault";
END_REGION

REGION Network 21: LH STOKER RUN (I 3.4)
   RUNG wire#powerrail
      Contact( "LH Stoker Run" )
      Coil( "DB100_WORK_BIT"."STAT33_LH Stoker Run" )
   END_RUNG
   // the same network as SCL:
   "DB100_WORK_BIT"."STAT33_LH Stoker Run" := "LH Stoker Run";
END_REGION

REGION Network 22: LH STOKER FAULT (I 3.5)
   RUNG wire#powerrail
      Contact( "LH Stoker Fault" )
      Coil( "DB100_WORK_BIT"."STAT35_LH Stoker Fault" )
   END_RUNG
   // the same network as SCL:
   "DB100_WORK_BIT"."STAT35_LH Stoker Fault" := "LH Stoker Fault";
END_REGION

REGION Network 23: RH STOKER RUN(I 3.6)
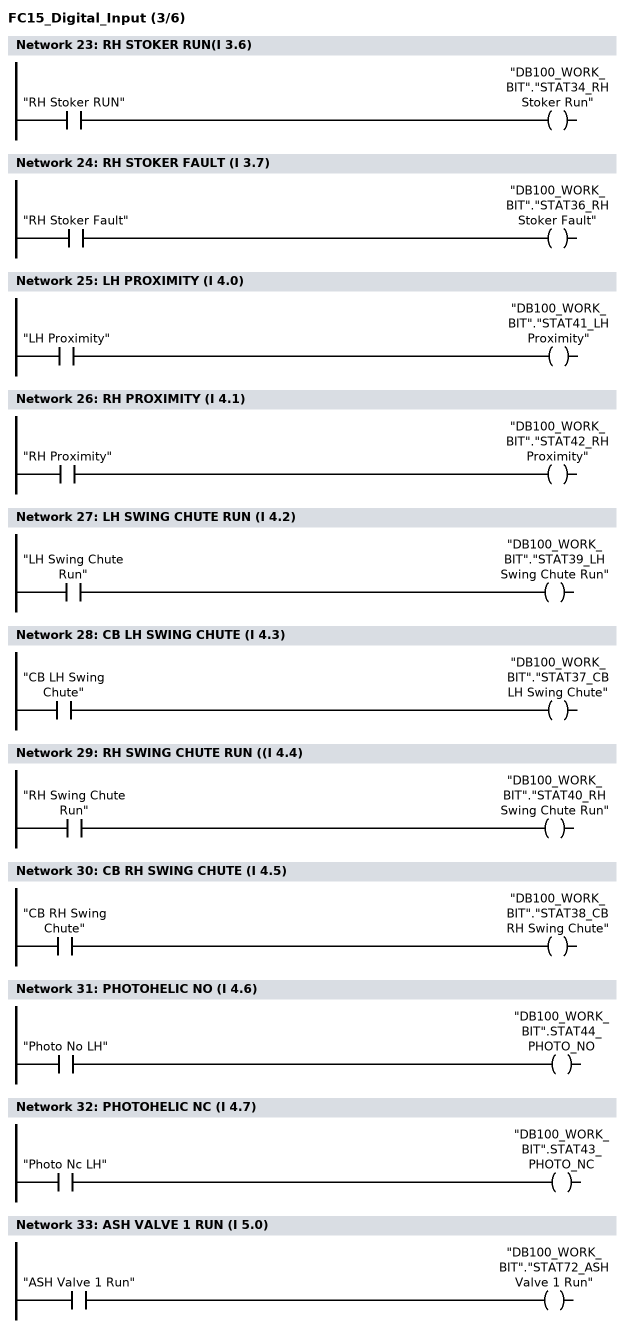
   RUNG wire#powerrail
      Contact( "RH Stoker RUN" )
      Coil( "DB100_WORK_BIT"."STAT34_RH Stoker Run" )
   END_RUNG
   // the same network as SCL:
   "DB100_WORK_BIT"."STAT34_RH Stoker Run" := "RH Stoker RUN";
END_REGION

REGION Network 24: RH STOKER FAULT (I 3.7)
   RUNG wire#powerrail
      Contact( "RH Stoker Fault" )
      Coil( "DB100_WORK_BIT"."STAT36_RH Stoker Fault" )
   END_RUNG
   // the same network as SCL:
   "DB100_WORK_BIT"."STAT36_RH Stoker Fault" := "RH Stoker Fault";
END_REGION

REGION Network 25: LH PROXIMITY (I 4.0)
   RUNG wire#powerrail
      Contact( "LH Proximity" )
      Coil( "DB100_WORK_BIT"."STAT41_LH Proximity" )
   END_RUNG
   // the same network as SCL:
   "DB100_WORK_BIT"."STAT41_LH Proximity" := "LH Proximity";
END_REGION

REGION Network 26: RH PROXIMITY (I 4.1)
   RUNG wire#powerrail
      Contact( "RH Proximity" )
      Coil( "DB100_WORK_BIT"."STAT42_RH Proximity" )
   END_RUNG
   // the same network as SCL:
   "DB100_WORK_BIT"."STAT42_RH Proximity" := "RH Proximity";
END_REGION

REGION Network 27: LH SWING CHUTE RUN (I 4.2)
   RUNG wire#powerrail
      Contact( "LH Swing Chute Run" )
      Coil( "DB100_WORK_BIT"."STAT39_LH Swing Chute Run" )
   END_RUNG
   // the same network as SCL:
   "DB100_WORK_BIT"."STAT39_LH Swing Chute Run" := "LH Swing Chute Run";
END_REGION

REGION Network 28: CB LH SWING CHUTE (I 4.3)
   RUNG wire#powerrail
      Contact( "CB LH Swing Chute" )
      Coil( "DB100_WORK_BIT"."STAT37_CB LH Swing Chute" )
   END_RUNG
   // the same network as SCL:
   "DB100_WORK_BIT"."STAT37_CB LH Swing Chute" := "CB LH Swing Chute";
END_REGION

REGION Network 29: RH SWING CHUTE RUN ((I 4.4)
   RUNG wire#powerrail
      Contact( "RH Swing Chute Run" )
      Coil( "DB100_WORK_BIT"."STAT40_RH Swing Chute Run" )
   END_RUNG
   // the same network as SCL:
   "DB100_WORK_BIT"."STAT40_RH Swing Chute Run" := "RH Swing Chute Run";
END_REGION

REGION Network 30: CB RH SWING CHUTE (I 4.5)
   RUNG wire#powerrail
      Contact( "CB RH Swing Chute" )
      Coil( "DB100_WORK_BIT"."STAT38_CB RH Swing Chute" )
   END_RUNG
   // the same network as SCL:
   "DB100_WORK_BIT"."STAT38_CB RH Swing Chute" := "CB RH Swing Chute";
END_REGION

REGION Network 31: PHOTOHELIC NO (I 4.6)
   RUNG wire#powerrail
      Contact( "Photo No LH" )
      Coil( "DB100_WORK_BIT".STAT44_PHOTO_NO )
   END_RUNG
   // the same network as SCL:
   "DB100_WORK_BIT".STAT44_PHOTO_NO := "Photo No LH";
END_REGION

REGION Network 32: PHOTOHELIC NC (I 4.7)
   RUNG wire#powerrail
      Contact( "Photo Nc LH" )
      Coil( "DB100_WORK_BIT".STAT43_PHOTO_NC )
   END_RUNG
   // the same network as SCL:
   "DB100_WORK_BIT".STAT43_PHOTO_NC := "Photo Nc LH";
END_REGION

REGION Network 33: ASH VALVE 1 RUN (I 5.0)
   RUNG wire#powerrail
      Contact( "ASH Valve 1 Run" )
      Coil( "DB100_WORK_BIT"."STAT72_ASH Valve 1 Run" )
   END_RUNG
   // the same network as SCL:
   "DB100_WORK_BIT"."STAT72_ASH Valve 1 Run" := "ASH Valve 1 Run";
END_REGION

REGION Network 34: CB ASH VALVE 1 (I 5.1)
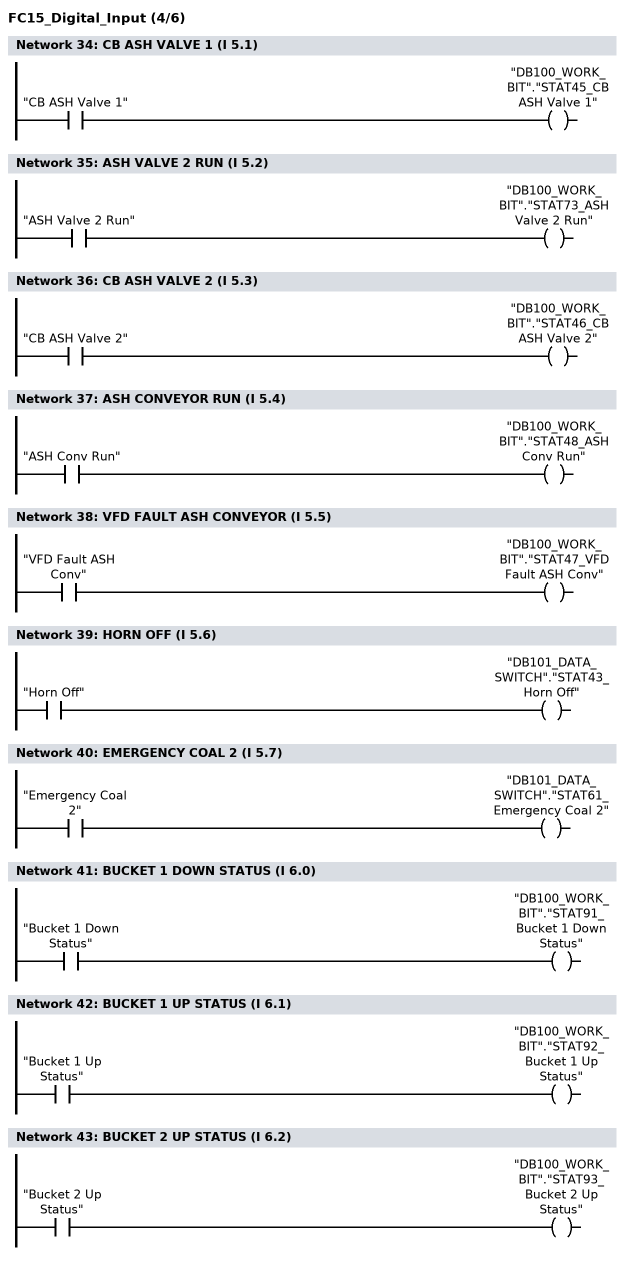
   RUNG wire#powerrail
      Contact( "CB ASH Valve 1" )
      Coil( "DB100_WORK_BIT"."STAT45_CB ASH Valve 1" )
   END_RUNG
   // the same network as SCL:
   "DB100_WORK_BIT"."STAT45_CB ASH Valve 1" := "CB ASH Valve 1";
END_REGION

REGION Network 35: ASH VALVE 2 RUN (I 5.2)
   RUNG wire#powerrail
      Contact( "ASH Valve 2 Run" )
      Coil( "DB100_WORK_BIT"."STAT73_ASH Valve 2 Run" )
   END_RUNG
   // the same network as SCL:
   "DB100_WORK_BIT"."STAT73_ASH Valve 2 Run" := "ASH Valve 2 Run";
END_REGION

REGION Network 36: CB ASH VALVE 2 (I 5.3)
   RUNG wire#powerrail
      Contact( "CB ASH Valve 2" )
      Coil( "DB100_WORK_BIT"."STAT46_CB ASH Valve 2" )
   END_RUNG
   // the same network as SCL:
   "DB100_WORK_BIT"."STAT46_CB ASH Valve 2" := "CB ASH Valve 2";
END_REGION

REGION Network 37: ASH CONVEYOR RUN (I 5.4)
   RUNG wire#powerrail
      Contact( "ASH Conv Run" )
      Coil( "DB100_WORK_BIT"."STAT48_ASH Conv Run" )
   END_RUNG
   // the same network as SCL:
   "DB100_WORK_BIT"."STAT48_ASH Conv Run" := "ASH Conv Run";
END_REGION

REGION Network 38: VFD FAULT ASH CONVEYOR (I 5.5)
   RUNG wire#powerrail
      Contact( "VFD Fault ASH Conv" )
      Coil( "DB100_WORK_BIT"."STAT47_VFD Fault ASH Conv" )
   END_RUNG
   // the same network as SCL:
   "DB100_WORK_BIT"."STAT47_VFD Fault ASH Conv" := "VFD Fault ASH Conv";
END_REGION

REGION Network 39: HORN OFF (I 5.6)
   RUNG wire#powerrail
      Contact( "Horn Off" )
      Coil( "DB101_DATA_SWITCH"."STAT43_Horn Off" )
   END_RUNG
   // the same network as SCL:
   "DB101_DATA_SWITCH"."STAT43_Horn Off" := "Horn Off";
END_REGION

REGION Network 40: EMERGENCY COAL 2 (I 5.7)
   RUNG wire#powerrail
      Contact( "Emergency Coal 2" )
      Coil( "DB101_DATA_SWITCH"."STAT61_Emergency Coal 2" )
   END_RUNG
   // the same network as SCL:
   "DB101_DATA_SWITCH"."STAT61_Emergency Coal 2" := "Emergency Coal 2";
END_REGION

REGION Network 41: BUCKET 1 DOWN STATUS (I 6.0)
   RUNG wire#powerrail
      Contact( "Bucket 1 Down Status" )
      Coil( "DB100_WORK_BIT"."STAT91_Bucket 1 Down Status" )
   END_RUNG
   // the same network as SCL:
   "DB100_WORK_BIT"."STAT91_Bucket 1 Down Status" := "Bucket 1 Down Status";
END_REGION

REGION Network 42: BUCKET 1 UP STATUS (I 6.1)
   RUNG wire#powerrail
      Contact( "Bucket 1 Up Status" )
      Coil( "DB100_WORK_BIT"."STAT92_Bucket 1 Up Status" )
   END_RUNG
   // the same network as SCL:
   "DB100_WORK_BIT"."STAT92_Bucket 1 Up Status" := "Bucket 1 Up Status";
END_REGION

REGION Network 43: BUCKET 2 UP STATUS (I 6.2)
   RUNG wire#powerrail
      Contact( "Bucket 2 Up Status" )
      Coil( "DB100_WORK_BIT"."STAT93_Bucket 2 Up Status" )
   END_RUNG
   // the same network as SCL:
   "DB100_WORK_BIT"."STAT93_Bucket 2 Up Status" := "Bucket 2 Up Status";
END_REGION

REGION Network 44: COAL EMPTY (I 6.3)
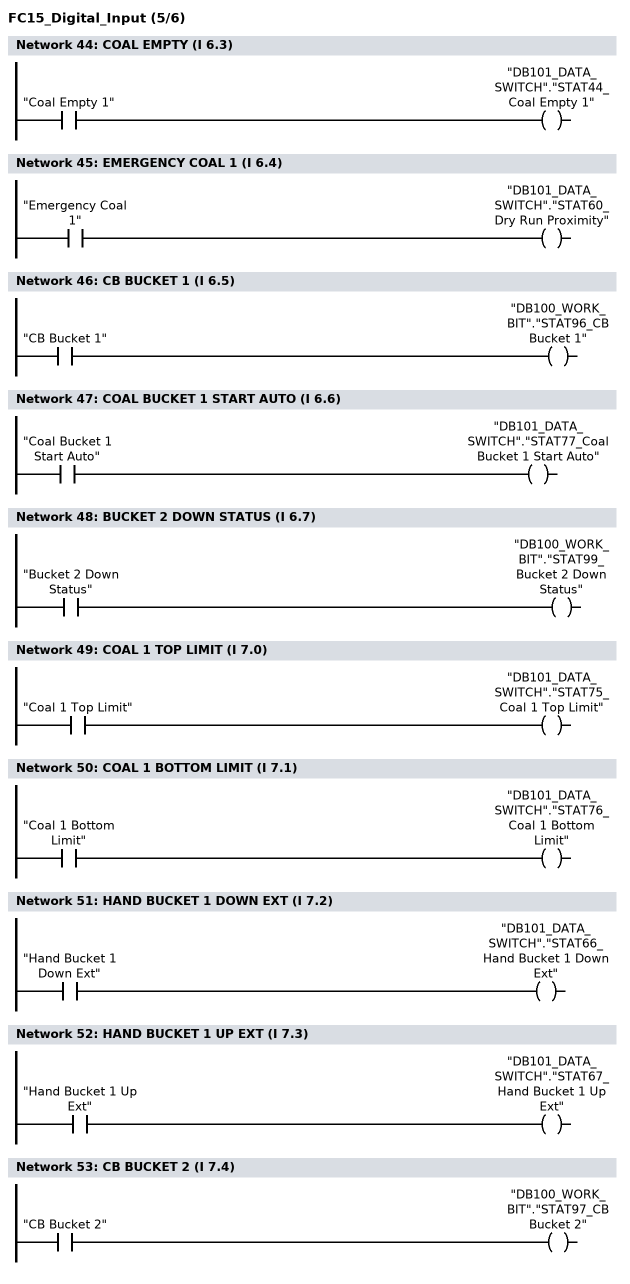
   RUNG wire#powerrail
      Contact( "Coal Empty 1" )
      Coil( "DB101_DATA_SWITCH"."STAT44_Coal Empty 1" )
   END_RUNG
   // the same network as SCL:
   "DB101_DATA_SWITCH"."STAT44_Coal Empty 1" := "Coal Empty 1";
END_REGION

REGION Network 45: EMERGENCY COAL 1 (I 6.4)
   RUNG wire#powerrail
      Contact( "Emergency Coal 1" )
      Coil( "DB101_DATA_SWITCH"."STAT60_Dry Run Proximity" )
   END_RUNG
   // the same network as SCL:
   "DB101_DATA_SWITCH"."STAT60_Dry Run Proximity" := "Emergency Coal 1";
END_REGION

REGION Network 46: CB BUCKET 1 (I 6.5)
   RUNG wire#powerrail
      Contact( "CB Bucket 1" )
      Coil( "DB100_WORK_BIT"."STAT96_CB Bucket 1" )
   END_RUNG
   // the same network as SCL:
   "DB100_WORK_BIT"."STAT96_CB Bucket 1" := "CB Bucket 1";
END_REGION

REGION Network 47: COAL BUCKET 1 START AUTO (I 6.6)
   RUNG wire#powerrail
      Contact( "Coal Bucket 1 Start Auto" )
      Coil( "DB101_DATA_SWITCH"."STAT77_Coal Bucket 1 Start Auto" )
   END_RUNG
   // the same network as SCL:
   "DB101_DATA_SWITCH"."STAT77_Coal Bucket 1 Start Auto" := "Coal Bucket 1 Start Auto";
END_REGION

REGION Network 48: BUCKET 2 DOWN STATUS (I 6.7)
   RUNG wire#powerrail
      Contact( "Bucket 2 Down Status" )
      Coil( "DB100_WORK_BIT"."STAT99_Bucket 2 Down Status" )
   END_RUNG
   // the same network as SCL:
   "DB100_WORK_BIT"."STAT99_Bucket 2 Down Status" := "Bucket 2 Down Status";
END_REGION

REGION Network 49: COAL 1 TOP LIMIT (I 7.0)
   RUNG wire#powerrail
      Contact( "Coal 1 Top Limit" )
      Coil( "DB101_DATA_SWITCH"."STAT75_Coal 1 Top Limit" )
   END_RUNG
   // the same network as SCL:
   "DB101_DATA_SWITCH"."STAT75_Coal 1 Top Limit" := "Coal 1 Top Limit";
END_REGION

REGION Network 50: COAL 1 BOTTOM LIMIT (I 7.1)
   RUNG wire#powerrail
      Contact( "Coal 1 Bottom Limit" )
      Coil( "DB101_DATA_SWITCH"."STAT76_Coal 1 Bottom Limit" )
   END_RUNG
   // the same network as SCL:
   "DB101_DATA_SWITCH"."STAT76_Coal 1 Bottom Limit" := "Coal 1 Bottom Limit";
END_REGION

REGION Network 51: HAND BUCKET 1 DOWN EXT (I 7.2)
   RUNG wire#powerrail
      Contact( "Hand Bucket 1 Down Ext" )
      Coil( "DB101_DATA_SWITCH"."STAT66_Hand Bucket 1 Down Ext" )
   END_RUNG
   // the same network as SCL:
   "DB101_DATA_SWITCH"."STAT66_Hand Bucket 1 Down Ext" := "Hand Bucket 1 Down Ext";
END_REGION

REGION Network 52: HAND BUCKET 1 UP EXT (I 7.3)
   RUNG wire#powerrail
      Contact( "Hand Bucket 1 Up Ext" )
      Coil( "DB101_DATA_SWITCH"."STAT67_Hand Bucket 1 Up Ext" )
   END_RUNG
   // the same network as SCL:
   "DB101_DATA_SWITCH"."STAT67_Hand Bucket 1 Up Ext" := "Hand Bucket 1 Up Ext";
END_REGION

REGION Network 53: CB BUCKET 2 (I 7.4)
   RUNG wire#powerrail
      Contact( "CB Bucket 2" )
      Coil( "DB100_WORK_BIT"."STAT97_CB Bucket 2" )
   END_RUNG
   // the same network as SCL:
   "DB100_WORK_BIT"."STAT97_CB Bucket 2" := "CB Bucket 2";
END_REGION

REGION Network 54: COAL BUCKET 2 START AUTO (I 7.5)
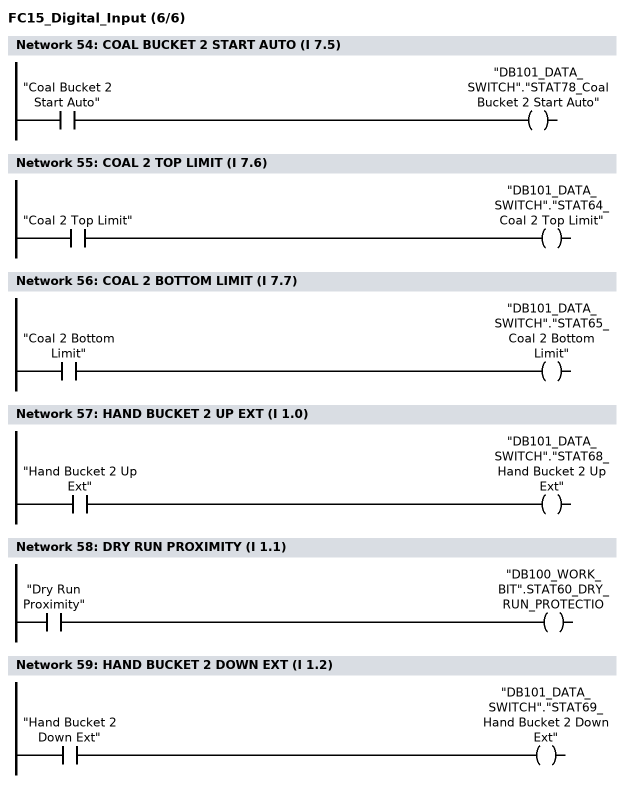
   RUNG wire#powerrail
      Contact( "Coal Bucket 2 Start Auto" )
      Coil( "DB101_DATA_SWITCH"."STAT78_Coal Bucket 2 Start Auto" )
   END_RUNG
   // the same network as SCL:
   "DB101_DATA_SWITCH"."STAT78_Coal Bucket 2 Start Auto" := "Coal Bucket 2 Start Auto";
END_REGION

REGION Network 55: COAL 2 TOP LIMIT (I 7.6)
   RUNG wire#powerrail
      Contact( "Coal 2 Top Limit" )
      Coil( "DB101_DATA_SWITCH"."STAT64_Coal 2 Top Limit" )
   END_RUNG
   // the same network as SCL:
   "DB101_DATA_SWITCH"."STAT64_Coal 2 Top Limit" := "Coal 2 Top Limit";
END_REGION

REGION Network 56: COAL 2 BOTTOM LIMIT (I 7.7)
   RUNG wire#powerrail
      Contact( "Coal 2 Bottom Limit" )
      Coil( "DB101_DATA_SWITCH"."STAT65_Coal 2 Bottom Limit" )
   END_RUNG
   // the same network as SCL:
   "DB101_DATA_SWITCH"."STAT65_Coal 2 Bottom Limit" := "Coal 2 Bottom Limit";
END_REGION

REGION Network 57: HAND BUCKET 2 UP EXT (I 1.0)
   RUNG wire#powerrail
      Contact( "Hand Bucket 2 Up Ext" )
      Coil( "DB101_DATA_SWITCH"."STAT68_Hand Bucket 2 Up Ext" )
   END_RUNG
   // the same network as SCL:
   "DB101_DATA_SWITCH"."STAT68_Hand Bucket 2 Up Ext" := "Hand Bucket 2 Up Ext";
END_REGION

REGION Network 58: DRY RUN PROXIMITY (I 1.1)
   RUNG wire#powerrail
      Contact( "Dry Run Proximity" )
      Coil( "DB100_WORK_BIT".STAT60_DRY_RUN_PROTECTIO )
   END_RUNG
   // the same network as SCL:
   "DB100_WORK_BIT".STAT60_DRY_RUN_PROTECTIO := "Dry Run Proximity";
END_REGION

REGION Network 59: HAND BUCKET 2 DOWN EXT (I 1.2)
   RUNG wire#powerrail
      Contact( "Hand Bucket 2 Down Ext" )
      Coil( "DB101_DATA_SWITCH"."STAT69_Hand Bucket 2 Down Ext" )
   END_RUNG
   // the same network as SCL:
   "DB101_DATA_SWITCH"."STAT69_Hand Bucket 2 Down Ext" := "Hand Bucket 2 Down Ext";
END_REGION
END_FUNCTION

FUNCTION "FC16_Digital_Output" : Void   // FC16, LAD
TITLE = Mapping Digital Output from DB 100
{ S7_Optimized_Access := 'TRUE' }
VERSION : 0.1
BEGIN

REGION Network 1: START FEED PUMP 1 (Q 0.0)
